BEGIN
   Zulauf_AR_Niv.Status.BA_Nrm := TRUE;
   Zulauf_AR_Niv.Status.BA_Frz := FALSE;
   Zulauf_AR_Niv.Status.BA_EW := FALSE;
   Zulauf_AR_Niv.Status.BA_Sim := FALSE;
   Zulauf_AR_Niv.Status.BA_Wart := FALSE;
   Zulauf_AR_Niv.Status.Frg_HH := FALSE;
   Zulauf_AR_Niv.Status.Frg_H := FALSE;
   Zulauf_AR_Niv.Status.Frg_L := FALSE;
   Zulauf_AR_Niv.Status.Frg_LL := FALSE;
   Zulauf_AR_Niv.Status.SB_MW_frz := FALSE;
   Zulauf_AR_Niv.Status.SB_MW_EW := FALSE;
   Zulauf_AR_Niv.Status.BM_MW_ok := TRUE;
   Zulauf_AR_Niv.Status.BM_MW_frz := FALSE;
   Zulauf_AR_Niv.Status.BM_MW_EW := FALSE;
   Zulauf_AR_Niv.Status.BM_MW_Sim := FALSE;
   Zulauf_AR_Niv.Status.BM_MW_nok := FALSE;
   Zulauf_AR_Niv.Status.BM_MW_zw := FALSE;
   Zulauf_AR_Niv.Status.GW_Sp_H := FALSE;
   Zulauf_AR_Niv.Status.GW_Sp_L := FALSE;
   Zulauf_AR_Niv.Status.Res_19 := FALSE;
   Zulauf_AR_Niv.Status.Res_26 := FALSE;
   Zulauf_AR_Niv.Status.Res_27 := FALSE;
   Zulauf_AR_Niv.Status.Res_28 := FALSE;
   Zulauf_AR_Niv.Status.Res_29 := FALSE;
   Zulauf_AR_Niv.Status.Res_30 := FALSE;
   Zulauf_AR_Niv.Status.Res_31 := FALSE;
   Zulauf_AR_Niv.Status.Res_32 := FALSE;
   Zulauf_AR_Niv.Status.Res_33 := FALSE;
   Zulauf_AR_Niv.Status.Res_34 := FALSE;
   Zulauf_AR_Niv.Status.BB_AutoOk := TRUE;
   Zulauf_AR_Niv.Status.BB_SS := FALSE;
   Zulauf_AR_Niv.Status.BB_SSnq := FALSE;
   Zulauf_AR_Niv.Stoerung.St_allg := FALSE;
   Zulauf_AR_Niv.Stoerung.St_4mA := FALSE;
   Zulauf_AR_Niv.Stoerung.St_OF := FALSE;
   Zulauf_AR_Niv.Stoerung.St_UF := FALSE;
   Zulauf_AR_Niv.Stoerung.St_Kom_DP := FALSE;
   Zulauf_AR_Niv.Stoerung.St_Kom_int := FALSE;
   Zulauf_AR_Niv.Stoerung.St_int := FALSE;
   Zulauf_AR_Niv.Stoerung.Res_7 := FALSE;
   Zulauf_AR_Niv.Stoerung.GW_HH := FALSE;
   Zulauf_AR_Niv.Stoerung.GW_H := FALSE;
   Zulauf_AR_Niv.Stoerung.GW_L := FALSE;
   Zulauf_AR_Niv.Stoerung.GW_LL := FALSE;
   Zulauf_AR_Niv.Stoerung.Res_12 := FALSE;
   Zulauf_AR_Niv.Stoerung.Res_13 := FALSE;
   Zulauf_AR_Niv.Stoerung.Res_14 := FALSE;
   Zulauf_AR_Niv.Stoerung.Res_15 := FALSE;
   Zulauf_AR_Niv.Stoerung.Res_16 := FALSE;
   Zulauf_AR_Niv.Stoerung.Res_17 := FALSE;
   Zulauf_AR_Niv.Stoerung.Res_18 := FALSE;
   Zulauf_AR_Niv.Stoerung.Res_19 := FALSE;
   Zulauf_AR_Niv.Stoerung.Res_20 := FALSE;
   Zulauf_AR_Niv.Stoerung.Res_21 := FALSE;
   Zulauf_AR_Niv.Stoerung.Res_22 := FALSE;
   Zulauf_AR_Niv.Stoerung.Res_23 := FALSE;
   Zulauf_AR_Niv.Stoerung.Res_24 := FALSE;
   Zulauf_AR_Niv.Stoerung.Res_25 := FALSE;
   Zulauf_AR_Niv.Stoerung.Res_26 := FALSE;
   Zulauf_AR_Niv.Stoerung.Res_27 := FALSE;
   Zulauf_AR_Niv.Stoerung.Res_28 := FALSE;
   Zulauf_AR_Niv.Stoerung.Res_29 := FALSE;
   Zulauf_AR_Niv.Stoerung.Res_30 := FALSE;
   Zulauf_AR_Niv.Stoerung.Res_31 := FALSE;
   Zulauf_AR_Niv.MW_akt := 21.85904;
   Zulauf_AR_Temp.Status.BA_Nrm := TRUE;
   Zulauf_AR_Temp.Status.BA_Frz := FALSE;
   Zulauf_AR_Temp.Status.BA_EW := FALSE;
   Zulauf_AR_Temp.Status.BA_Sim := FALSE;
   Zulauf_AR_Temp.Status.BA_Wart := FALSE;
   Zulauf_AR_Temp.Status.Frg_HH := FALSE;
   Zulauf_AR_Temp.Status.Frg_H := FALSE;
   Zulauf_AR_Temp.Status.Frg_L := FALSE;
   Zulauf_AR_Temp.Status.Frg_LL := FALSE;
   Zulauf_AR_Temp.Status.SB_MW_frz := FALSE;
   Zulauf_AR_Temp.Status.SB_MW_EW := FALSE;
   Zulauf_AR_Temp.Status.BM_MW_ok := TRUE;
   Zulauf_AR_Temp.Status.BM_MW_frz := FALSE;
   Zulauf_AR_Temp.Status.BM_MW_EW := FALSE;
   Zulauf_AR_Temp.Status.BM_MW_Sim := FALSE;
   Zulauf_AR_Temp.Status.BM_MW_nok := FALSE;
   Zulauf_AR_Temp.Status.BM_MW_zw := FALSE;
   Zulauf_AR_Temp.Status.GW_Sp_H := FALSE;
   Zulauf_AR_Temp.Status.GW_Sp_L := FALSE;
   Zulauf_AR_Temp.Status.Res_19 := FALSE;
   Zulauf_AR_Temp.Status.Res_26 := FALSE;
   Zulauf_AR_Temp.Status.Res_27 := FALSE;
   Zulauf_AR_Temp.Status.Res_28 := FALSE;
   Zulauf_AR_Temp.Status.Res_29 := FALSE;
   Zulauf_AR_Temp.Status.Res_30 := FALSE;
   Zulauf_AR_Temp.Status.Res_31 := FALSE;
   Zulauf_AR_Temp.Status.Res_32 := FALSE;
   Zulauf_AR_Temp.Status.Res_33 := FALSE;
   Zulauf_AR_Temp.Status.Res_34 := FALSE;
   Zulauf_AR_Temp.Status.BB_AutoOk := TRUE;
   Zulauf_AR_Temp.Status.BB_SS := FALSE;
   Zulauf_AR_Temp.Status.BB_SSnq := FALSE;
   Zulauf_AR_Temp.Stoerung.St_allg := FALSE;
   Zulauf_AR_Temp.Stoerung.St_4mA := FALSE;
   Zulauf_AR_Temp.Stoerung.St_OF := FALSE;
   Zulauf_AR_Temp.Stoerung.St_UF := FALSE;
   Zulauf_AR_Temp.Stoerung.St_Kom_DP := FALSE;
   Zulauf_AR_Temp.Stoerung.St_Kom_int := FALSE;
   Zulauf_AR_Temp.Stoerung.St_int := FALSE;
   Zulauf_AR_Temp.Stoerung.Res_7 := FALSE;
   Zulauf_AR_Temp.Stoerung.GW_HH := FALSE;
   Zulauf_AR_Temp.Stoerung.GW_H := FALSE;
   Zulauf_AR_Temp.Stoerung.GW_L := FALSE;
   Zulauf_AR_Temp.Stoerung.GW_LL := FALSE;
   Zulauf_AR_Temp.Stoerung.Res_12 := FALSE;
   Zulauf_AR_Temp.Stoerung.Res_13 := FALSE;
   Zulauf_AR_Temp.Stoerung.Res_14 := FALSE;
   Zulauf_AR_Temp.Stoerung.Res_15 := FALSE;
   Zulauf_AR_Temp.Stoerung.Res_16 := FALSE;
   Zulauf_AR_Temp.Stoerung.Res_17 := FALSE;
   Zulauf_AR_Temp.Stoerung.Res_18 := FALSE;
   Zulauf_AR_Temp.Stoerung.Res_19 := FALSE;
   Zulauf_AR_Temp.Stoerung.Res_20 := FALSE;
   Zulauf_AR_Temp.Stoerung.Res_21 := FALSE;
   Zulauf_AR_Temp.Stoerung.Res_22 := FALSE;
   Zulauf_AR_Temp.Stoerung.Res_23 := FALSE;
   Zulauf_AR_Temp.Stoerung.Res_24 := FALSE;
   Zulauf_AR_Temp.Stoerung.Res_25 := FALSE;
   Zulauf_AR_Temp.Stoerung.Res_26 := FALSE;
   Zulauf_AR_Temp.Stoerung.Res_27 := FALSE;
   Zulauf_AR_Temp.Stoerung.Res_28 := FALSE;
   Zulauf_AR_Temp.Stoerung.Res_29 := FALSE;
   Zulauf_AR_Temp.Stoerung.Res_30 := FALSE;
   Zulauf_AR_Temp.Stoerung.Res_31 := FALSE;
   Zulauf_AR_Temp.MW_akt := 0.0;
   Zulauf_AR_DF.Status.BA_Nrm := TRUE;
   Zulauf_AR_DF.Status.BA_Frz := FALSE;
   Zulauf_AR_DF.Status.BA_EW := FALSE;
   Zulauf_AR_DF.Status.BA_Sim := FALSE;
   Zulauf_AR_DF.Status.BA_Wart := FALSE;
   Zulauf_AR_DF.Status.Frg_HH := FALSE;
   Zulauf_AR_DF.Status.Frg_H := FALSE;
   Zulauf_AR_DF.Status.Frg_L := FALSE;
   Zulauf_AR_DF.Status.Frg_LL := FALSE;
   Zulauf_AR_DF.Status.SB_MW_frz := FALSE;
   Zulauf_AR_DF.Status.SB_MW_EW := FALSE;
   Zulauf_AR_DF.Status.BM_MW_ok := FALSE;
   Zulauf_AR_DF.Status.BM_MW_frz := TRUE;
   Zulauf_AR_DF.Status.BM_MW_EW := FALSE;
   Zulauf_AR_DF.Status.BM_MW_Sim := FALSE;
   Zulauf_AR_DF.Status.BM_MW_nok := TRUE;
   Zulauf_AR_DF.Status.BM_MW_zw := FALSE;
   Zulauf_AR_DF.Status.GW_Sp_H := FALSE;
   Zulauf_AR_DF.Status.GW_Sp_L := FALSE;
   Zulauf_AR_DF.Status.Res_19 := FALSE;
   Zulauf_AR_DF.Status.Res_26 := FALSE;
   Zulauf_AR_DF.Status.Res_27 := FALSE;
   Zulauf_AR_DF.Status.Res_28 := FALSE;
   Zulauf_AR_DF.Status.Res_29 := FALSE;
   Zulauf_AR_DF.Status.Res_30 := FALSE;
   Zulauf_AR_DF.Status.Res_31 := FALSE;
   Zulauf_AR_DF.Status.Res_32 := FALSE;
   Zulauf_AR_DF.Status.Res_33 := FALSE;
   Zulauf_AR_DF.Status.Res_34 := FALSE;
   Zulauf_AR_DF.Status.BB_AutoOk := FALSE;
   Zulauf_AR_DF.Status.BB_SS := TRUE;
   Zulauf_AR_DF.Status.BB_SSnq := FALSE;
   Zulauf_AR_DF.Stoerung.St_allg := FALSE;
   Zulauf_AR_DF.Stoerung.St_4mA := TRUE;
   Zulauf_AR_DF.Stoerung.St_OF := FALSE;
   Zulauf_AR_DF.Stoerung.St_UF := TRUE;
   Zulauf_AR_DF.Stoerung.St_Kom_DP := FALSE;
   Zulauf_AR_DF.Stoerung.St_Kom_int := FALSE;
   Zulauf_AR_DF.Stoerung.St_int := FALSE;
   Zulauf_AR_DF.Stoerung.Res_7 := FALSE;
   Zulauf_AR_DF.Stoerung.GW_HH := FALSE;
   Zulauf_AR_DF.Stoerung.GW_H := FALSE;
   Zulauf_AR_DF.Stoerung.GW_L := FALSE;
   Zulauf_AR_DF.Stoerung.GW_LL := FALSE;
   Zulauf_AR_DF.Stoerung.Res_12 := FALSE;
   Zulauf_AR_DF.Stoerung.Res_13 := FALSE;
   Zulauf_AR_DF.Stoerung.Res_14 := FALSE;
   Zulauf_AR_DF.Stoerung.Res_15 := FALSE;
   Zulauf_AR_DF.Stoerung.Res_16 := FALSE;
   Zulauf_AR_DF.Stoerung.Res_17 := FALSE;
   Zulauf_AR_DF.Stoerung.Res_18 := FALSE;
   Zulauf_AR_DF.Stoerung.Res_19 := FALSE;
   Zulauf_AR_DF.Stoerung.Res_20 := FALSE;
   Zulauf_AR_DF.Stoerung.Res_21 := FALSE;
   Zulauf_AR_DF.Stoerung.Res_22 := FALSE;
   Zulauf_AR_DF.Stoerung.Res_23 := FALSE;
   Zulauf_AR_DF.Stoerung.Res_24 := FALSE;
   Zulauf_AR_DF.Stoerung.Res_25 := FALSE;
   Zulauf_AR_DF.Stoerung.Res_26 := FALSE;
   Zulauf_AR_DF.Stoerung.Res_27 := FALSE;
   Zulauf_AR_DF.Stoerung.Res_28 := FALSE;
   Zulauf_AR_DF.Stoerung.Res_29 := FALSE;
   Zulauf_AR_DF.Stoerung.Res_30 := FALSE;
   Zulauf_AR_DF.Stoerung.Res_31 := FALSE;
   Zulauf_AR_DF.MW_akt := 0.0;
   BB1_AS1_SS.Status.BA_Nrm := TRUE;
   BB1_AS1_SS.Status.BA_Frz := FALSE;
   BB1_AS1_SS.Status.BA_EW := FALSE;
   BB1_AS1_SS.Status.BA_Sim := FALSE;
   BB1_AS1_SS.Status.BA_Wart := FALSE;
   BB1_AS1_SS.Status.Frg_HH := FALSE;
   BB1_AS1_SS.Status.Frg_H := FALSE;
   BB1_AS1_SS.Status.Frg_L := FALSE;
   BB1_AS1_SS.Status.Frg_LL := FALSE;
   BB1_AS1_SS.Status.SB_MW_frz := FALSE;
   BB1_AS1_SS.Status.SB_MW_EW := FALSE;
   BB1_AS1_SS.Status.BM_MW_ok := TRUE;
   BB1_AS1_SS.Status.BM_MW_frz := FALSE;
   BB1_AS1_SS.Status.BM_MW_EW := FALSE;
   BB1_AS1_SS.Status.BM_MW_Sim := FALSE;
   BB1_AS1_SS.Status.BM_MW_nok := FALSE;
   BB1_AS1_SS.Status.BM_MW_zw := FALSE;
   BB1_AS1_SS.Status.GW_Sp_H := FALSE;
   BB1_AS1_SS.Status.GW_Sp_L := FALSE;
   BB1_AS1_SS.Status.Res_19 := FALSE;
   BB1_AS1_SS.Status.Res_26 := FALSE;
   BB1_AS1_SS.Status.Res_27 := FALSE;
   BB1_AS1_SS.Status.Res_28 := FALSE;
   BB1_AS1_SS.Status.Res_29 := FALSE;
   BB1_AS1_SS.Status.Res_30 := FALSE;
   BB1_AS1_SS.Status.Res_31 := FALSE;
   BB1_AS1_SS.Status.Res_32 := FALSE;
   BB1_AS1_SS.Status.Res_33 := FALSE;
   BB1_AS1_SS.Status.Res_34 := FALSE;
   BB1_AS1_SS.Status.BB_AutoOk := TRUE;
   BB1_AS1_SS.Status.BB_SS := FALSE;
   BB1_AS1_SS.Status.BB_SSnq := FALSE;
   BB1_AS1_SS.Stoerung.St_allg := FALSE;
   BB1_AS1_SS.Stoerung.St_4mA := FALSE;
   BB1_AS1_SS.Stoerung.St_OF := FALSE;
   BB1_AS1_SS.Stoerung.St_UF := FALSE;
   BB1_AS1_SS.Stoerung.St_Kom_DP := FALSE;
   BB1_AS1_SS.Stoerung.St_Kom_int := FALSE;
   BB1_AS1_SS.Stoerung.St_int := FALSE;
   BB1_AS1_SS.Stoerung.Res_7 := FALSE;
   BB1_AS1_SS.Stoerung.GW_HH := FALSE;
   BB1_AS1_SS.Stoerung.GW_H := FALSE;
   BB1_AS1_SS.Stoerung.GW_L := FALSE;
   BB1_AS1_SS.Stoerung.GW_LL := FALSE;
   BB1_AS1_SS.Stoerung.Res_12 := FALSE;
   BB1_AS1_SS.Stoerung.Res_13 := FALSE;
   BB1_AS1_SS.Stoerung.Res_14 := FALSE;
   BB1_AS1_SS.Stoerung.Res_15 := FALSE;
   BB1_AS1_SS.Stoerung.Res_16 := FALSE;
   BB1_AS1_SS.Stoerung.Res_17 := FALSE;
   BB1_AS1_SS.Stoerung.Res_18 := FALSE;
   BB1_AS1_SS.Stoerung.Res_19 := FALSE;
   BB1_AS1_SS.Stoerung.Res_20 := FALSE;
   BB1_AS1_SS.Stoerung.Res_21 := FALSE;
   BB1_AS1_SS.Stoerung.Res_22 := FALSE;
   BB1_AS1_SS.Stoerung.Res_23 := FALSE;
   BB1_AS1_SS.Stoerung.Res_24 := FALSE;
   BB1_AS1_SS.Stoerung.Res_25 := FALSE;
   BB1_AS1_SS.Stoerung.Res_26 := FALSE;
   BB1_AS1_SS.Stoerung.Res_27 := FALSE;
   BB1_AS1_SS.Stoerung.Res_28 := FALSE;
   BB1_AS1_SS.Stoerung.Res_29 := FALSE;
   BB1_AS1_SS.Stoerung.Res_30 := FALSE;
   BB1_AS1_SS.Stoerung.Res_31 := FALSE;
   BB1_AS1_SS.MW_akt := 0.0;
   BB1_AS2_SS.Status.BA_Nrm := TRUE;
   BB1_AS2_SS.Status.BA_Frz := FALSE;
   BB1_AS2_SS.Status.BA_EW := FALSE;
   BB1_AS2_SS.Status.BA_Sim := FALSE;
   BB1_AS2_SS.Status.BA_Wart := FALSE;
   BB1_AS2_SS.Status.Frg_HH := FALSE;
   BB1_AS2_SS.Status.Frg_H := FALSE;
   BB1_AS2_SS.Status.Frg_L := FALSE;
   BB1_AS2_SS.Status.Frg_LL := FALSE;
   BB1_AS2_SS.Status.SB_MW_frz := FALSE;
   BB1_AS2_SS.Status.SB_MW_EW := FALSE;
   BB1_AS2_SS.Status.BM_MW_ok := TRUE;
   BB1_AS2_SS.Status.BM_MW_frz := FALSE;
   BB1_AS2_SS.Status.BM_MW_EW := FALSE;
   BB1_AS2_SS.Status.BM_MW_Sim := FALSE;
   BB1_AS2_SS.Status.BM_MW_nok := FALSE;
   BB1_AS2_SS.Status.BM_MW_zw := FALSE;
   BB1_AS2_SS.Status.GW_Sp_H := FALSE;
   BB1_AS2_SS.Status.GW_Sp_L := FALSE;
   BB1_AS2_SS.Status.Res_19 := FALSE;
   BB1_AS2_SS.Status.Res_26 := FALSE;
   BB1_AS2_SS.Status.Res_27 := FALSE;
   BB1_AS2_SS.Status.Res_28 := FALSE;
   BB1_AS2_SS.Status.Res_29 := FALSE;
   BB1_AS2_SS.Status.Res_30 := FALSE;
   BB1_AS2_SS.Status.Res_31 := FALSE;
   BB1_AS2_SS.Status.Res_32 := FALSE;
   BB1_AS2_SS.Status.Res_33 := FALSE;
   BB1_AS2_SS.Status.Res_34 := FALSE;
   BB1_AS2_SS.Status.BB_AutoOk := TRUE;
   BB1_AS2_SS.Status.BB_SS := FALSE;
   BB1_AS2_SS.Status.BB_SSnq := FALSE;
   BB1_AS2_SS.Stoerung.St_allg := FALSE;
   BB1_AS2_SS.Stoerung.St_4mA := FALSE;
   BB1_AS2_SS.Stoerung.St_OF := FALSE;
   BB1_AS2_SS.Stoerung.St_UF := FALSE;
   BB1_AS2_SS.Stoerung.St_Kom_DP := FALSE;
   BB1_AS2_SS.Stoerung.St_Kom_int := FALSE;
   BB1_AS2_SS.Stoerung.St_int := FALSE;
   BB1_AS2_SS.Stoerung.Res_7 := FALSE;
   BB1_AS2_SS.Stoerung.GW_HH := FALSE;
   BB1_AS2_SS.Stoerung.GW_H := FALSE;
   BB1_AS2_SS.Stoerung.GW_L := FALSE;
   BB1_AS2_SS.Stoerung.GW_LL := FALSE;
   BB1_AS2_SS.Stoerung.Res_12 := FALSE;
   BB1_AS2_SS.Stoerung.Res_13 := FALSE;
   BB1_AS2_SS.Stoerung.Res_14 := FALSE;
   BB1_AS2_SS.Stoerung.Res_15 := FALSE;
   BB1_AS2_SS.Stoerung.Res_16 := FALSE;
   BB1_AS2_SS.Stoerung.Res_17 := FALSE;
   BB1_AS2_SS.Stoerung.Res_18 := FALSE;
   BB1_AS2_SS.Stoerung.Res_19 := FALSE;
   BB1_AS2_SS.Stoerung.Res_20 := FALSE;
   BB1_AS2_SS.Stoerung.Res_21 := FALSE;
   BB1_AS2_SS.Stoerung.Res_22 := FALSE;
   BB1_AS2_SS.Stoerung.Res_23 := FALSE;
   BB1_AS2_SS.Stoerung.Res_24 := FALSE;
   BB1_AS2_SS.Stoerung.Res_25 := FALSE;
   BB1_AS2_SS.Stoerung.Res_26 := FALSE;
   BB1_AS2_SS.Stoerung.Res_27 := FALSE;
   BB1_AS2_SS.Stoerung.Res_28 := FALSE;
   BB1_AS2_SS.Stoerung.Res_29 := FALSE;
   BB1_AS2_SS.Stoerung.Res_30 := FALSE;
   BB1_AS2_SS.Stoerung.Res_31 := FALSE;
   BB1_AS2_SS.MW_akt := 76.62236;
   BB2_AS1_SS.Status.BA_Nrm := TRUE;
   BB2_AS1_SS.Status.BA_Frz := FALSE;
   BB2_AS1_SS.Status.BA_EW := FALSE;
   BB2_AS1_SS.Status.BA_Sim := FALSE;
   BB2_AS1_SS.Status.BA_Wart := FALSE;
   BB2_AS1_SS.Status.Frg_HH := FALSE;
   BB2_AS1_SS.Status.Frg_H := FALSE;
   BB2_AS1_SS.Status.Frg_L := FALSE;
   BB2_AS1_SS.Status.Frg_LL := FALSE;
   BB2_AS1_SS.Status.SB_MW_frz := FALSE;
   BB2_AS1_SS.Status.SB_MW_EW := FALSE;
   BB2_AS1_SS.Status.BM_MW_ok := TRUE;
   BB2_AS1_SS.Status.BM_MW_frz := FALSE;
   BB2_AS1_SS.Status.BM_MW_EW := FALSE;
   BB2_AS1_SS.Status.BM_MW_Sim := FALSE;
   BB2_AS1_SS.Status.BM_MW_nok := FALSE;
   BB2_AS1_SS.Status.BM_MW_zw := FALSE;
   BB2_AS1_SS.Status.GW_Sp_H := FALSE;
   BB2_AS1_SS.Status.GW_Sp_L := FALSE;
   BB2_AS1_SS.Status.Res_19 := FALSE;
   BB2_AS1_SS.Status.Res_26 := FALSE;
   BB2_AS1_SS.Status.Res_27 := FALSE;
   BB2_AS1_SS.Status.Res_28 := FALSE;
   BB2_AS1_SS.Status.Res_29 := FALSE;
   BB2_AS1_SS.Status.Res_30 := FALSE;
   BB2_AS1_SS.Status.Res_31 := FALSE;
   BB2_AS1_SS.Status.Res_32 := FALSE;
   BB2_AS1_SS.Status.Res_33 := FALSE;
   BB2_AS1_SS.Status.Res_34 := FALSE;
   BB2_AS1_SS.Status.BB_AutoOk := TRUE;
   BB2_AS1_SS.Status.BB_SS := FALSE;
   BB2_AS1_SS.Status.BB_SSnq := FALSE;
   BB2_AS1_SS.Stoerung.St_allg := FALSE;
   BB2_AS1_SS.Stoerung.St_4mA := FALSE;
   BB2_AS1_SS.Stoerung.St_OF := FALSE;
   BB2_AS1_SS.Stoerung.St_UF := FALSE;
   BB2_AS1_SS.Stoerung.St_Kom_DP := FALSE;
   BB2_AS1_SS.Stoerung.St_Kom_int := FALSE;
   BB2_AS1_SS.Stoerung.St_int := FALSE;
   BB2_AS1_SS.Stoerung.Res_7 := FALSE;
   BB2_AS1_SS.Stoerung.GW_HH := FALSE;
   BB2_AS1_SS.Stoerung.GW_H := FALSE;
   BB2_AS1_SS.Stoerung.GW_L := FALSE;
   BB2_AS1_SS.Stoerung.GW_LL := FALSE;
   BB2_AS1_SS.Stoerung.Res_12 := FALSE;
   BB2_AS1_SS.Stoerung.Res_13 := FALSE;
   BB2_AS1_SS.Stoerung.Res_14 := FALSE;
   BB2_AS1_SS.Stoerung.Res_15 := FALSE;
   BB2_AS1_SS.Stoerung.Res_16 := FALSE;
   BB2_AS1_SS.Stoerung.Res_17 := FALSE;
   BB2_AS1_SS.Stoerung.Res_18 := FALSE;
   BB2_AS1_SS.Stoerung.Res_19 := FALSE;
   BB2_AS1_SS.Stoerung.Res_20 := FALSE;
   BB2_AS1_SS.Stoerung.Res_21 := FALSE;
   BB2_AS1_SS.Stoerung.Res_22 := FALSE;
   BB2_AS1_SS.Stoerung.Res_23 := FALSE;
   BB2_AS1_SS.Stoerung.Res_24 := FALSE;
   BB2_AS1_SS.Stoerung.Res_25 := FALSE;
   BB2_AS1_SS.Stoerung.Res_26 := FALSE;
   BB2_AS1_SS.Stoerung.Res_27 := FALSE;
   BB2_AS1_SS.Stoerung.Res_28 := FALSE;
   BB2_AS1_SS.Stoerung.Res_29 := FALSE;
   BB2_AS1_SS.Stoerung.Res_30 := FALSE;
   BB2_AS1_SS.Stoerung.Res_31 := FALSE;
   BB2_AS1_SS.MW_akt := 0.05018311;
   BB2_AS2_SS.Status.BA_Nrm := TRUE;
   BB2_AS2_SS.Status.BA_Frz := FALSE;
   BB2_AS2_SS.Status.BA_EW := FALSE;
   BB2_AS2_SS.Status.BA_Sim := FALSE;
   BB2_AS2_SS.Status.BA_Wart := FALSE;
   BB2_AS2_SS.Status.Frg_HH := FALSE;
   BB2_AS2_SS.Status.Frg_H := FALSE;
   BB2_AS2_SS.Status.Frg_L := FALSE;
   BB2_AS2_SS.Status.Frg_LL := FALSE;
   BB2_AS2_SS.Status.SB_MW_frz := FALSE;
   BB2_AS2_SS.Status.SB_MW_EW := FALSE;
   BB2_AS2_SS.Status.BM_MW_ok := TRUE;
   BB2_AS2_SS.Status.BM_MW_frz := FALSE;
   BB2_AS2_SS.Status.BM_MW_EW := FALSE;
   BB2_AS2_SS.Status.BM_MW_Sim := FALSE;
   BB2_AS2_SS.Status.BM_MW_nok := FALSE;
   BB2_AS2_SS.Status.BM_MW_zw := FALSE;
   BB2_AS2_SS.Status.GW_Sp_H := FALSE;
   BB2_AS2_SS.Status.GW_Sp_L := FALSE;
   BB2_AS2_SS.Status.Res_19 := FALSE;
   BB2_AS2_SS.Status.Res_26 := FALSE;
   BB2_AS2_SS.Status.Res_27 := FALSE;
   BB2_AS2_SS.Status.Res_28 := FALSE;
   BB2_AS2_SS.Status.Res_29 := FALSE;
   BB2_AS2_SS.Status.Res_30 := FALSE;
   BB2_AS2_SS.Status.Res_31 := FALSE;
   BB2_AS2_SS.Status.Res_32 := FALSE;
   BB2_AS2_SS.Status.Res_33 := FALSE;
   BB2_AS2_SS.Status.Res_34 := FALSE;
   BB2_AS2_SS.Status.BB_AutoOk := TRUE;
   BB2_AS2_SS.Status.BB_SS := FALSE;
   BB2_AS2_SS.Status.BB_SSnq := FALSE;
   BB2_AS2_SS.Stoerung.St_allg := FALSE;
   BB2_AS2_SS.Stoerung.St_4mA := FALSE;
   BB2_AS2_SS.Stoerung.St_OF := FALSE;
   BB2_AS2_SS.Stoerung.St_UF := FALSE;
   BB2_AS2_SS.Stoerung.St_Kom_DP := FALSE;
   BB2_AS2_SS.Stoerung.St_Kom_int := FALSE;
   BB2_AS2_SS.Stoerung.St_int := FALSE;
   BB2_AS2_SS.Stoerung.Res_7 := FALSE;
   BB2_AS2_SS.Stoerung.GW_HH := FALSE;
   BB2_AS2_SS.Stoerung.GW_H := FALSE;
   BB2_AS2_SS.Stoerung.GW_L := FALSE;
   BB2_AS2_SS.Stoerung.GW_LL := FALSE;
   BB2_AS2_SS.Stoerung.Res_12 := FALSE;
   BB2_AS2_SS.Stoerung.Res_13 := FALSE;
   BB2_AS2_SS.Stoerung.Res_14 := FALSE;
   BB2_AS2_SS.Stoerung.Res_15 := FALSE;
   BB2_AS2_SS.Stoerung.Res_16 := FALSE;
   BB2_AS2_SS.Stoerung.Res_17 := FALSE;
   BB2_AS2_SS.Stoerung.Res_18 := FALSE;
   BB2_AS2_SS.Stoerung.Res_19 := FALSE;
   BB2_AS2_SS.Stoerung.Res_20 := FALSE;
   BB2_AS2_SS.Stoerung.Res_21 := FALSE;
   BB2_AS2_SS.Stoerung.Res_22 := FALSE;
   BB2_AS2_SS.Stoerung.Res_23 := FALSE;
   BB2_AS2_SS.Stoerung.Res_24 := FALSE;
   BB2_AS2_SS.Stoerung.Res_25 := FALSE;
   BB2_AS2_SS.Stoerung.Res_26 := FALSE;
   BB2_AS2_SS.Stoerung.Res_27 := FALSE;
   BB2_AS2_SS.Stoerung.Res_28 := FALSE;
   BB2_AS2_SS.Stoerung.Res_29 := FALSE;
   BB2_AS2_SS.Stoerung.Res_30 := FALSE;
   BB2_AS2_SS.Stoerung.Res_31 := FALSE;
   BB2_AS2_SS.MW_akt := 0.140151;
   BB1_O2.Status.BA_Nrm := TRUE;
   BB1_O2.Status.BA_Frz := FALSE;
   BB1_O2.Status.BA_EW := FALSE;
   BB1_O2.Status.BA_Sim := FALSE;
   BB1_O2.Status.BA_Wart := FALSE;
   BB1_O2.Status.Frg_HH := FALSE;
   BB1_O2.Status.Frg_H := FALSE;
   BB1_O2.Status.Frg_L := FALSE;
   BB1_O2.Status.Frg_LL := TRUE;
   BB1_O2.Status.SB_MW_frz := FALSE;
   BB1_O2.Status.SB_MW_EW := FALSE;
   BB1_O2.Status.BM_MW_ok := TRUE;
   BB1_O2.Status.BM_MW_frz := FALSE;
   BB1_O2.Status.BM_MW_EW := FALSE;
   BB1_O2.Status.BM_MW_Sim := FALSE;
   BB1_O2.Status.BM_MW_nok := FALSE;
   BB1_O2.Status.BM_MW_zw := FALSE;
   BB1_O2.Status.GW_Sp_H := FALSE;
   BB1_O2.Status.GW_Sp_L := FALSE;
   BB1_O2.Status.Res_19 := FALSE;
   BB1_O2.Status.Res_26 := FALSE;
   BB1_O2.Status.Res_27 := FALSE;
   BB1_O2.Status.Res_28 := FALSE;
   BB1_O2.Status.Res_29 := FALSE;
   BB1_O2.Status.Res_30 := FALSE;
   BB1_O2.Status.Res_31 := FALSE;
   BB1_O2.Status.Res_32 := FALSE;
   BB1_O2.Status.Res_33 := FALSE;
   BB1_O2.Status.Res_34 := FALSE;
   BB1_O2.Status.BB_AutoOk := TRUE;
   BB1_O2.Status.BB_SS := FALSE;
   BB1_O2.Status.BB_SSnq := FALSE;
   BB1_O2.Stoerung.St_allg := FALSE;
   BB1_O2.Stoerung.St_4mA := FALSE;
   BB1_O2.Stoerung.St_OF := FALSE;
   BB1_O2.Stoerung.St_UF := FALSE;
   BB1_O2.Stoerung.St_Kom_DP := FALSE;
   BB1_O2.Stoerung.St_Kom_int := FALSE;
   BB1_O2.Stoerung.St_int := FALSE;
   BB1_O2.Stoerung.Res_7 := FALSE;
   BB1_O2.Stoerung.GW_HH := FALSE;
   BB1_O2.Stoerung.GW_H := FALSE;
   BB1_O2.Stoerung.GW_L := FALSE;
   BB1_O2.Stoerung.GW_LL := FALSE;
   BB1_O2.Stoerung.Res_12 := FALSE;
   BB1_O2.Stoerung.Res_13 := FALSE;
   BB1_O2.Stoerung.Res_14 := FALSE;
   BB1_O2.Stoerung.Res_15 := FALSE;
   BB1_O2.Stoerung.Res_16 := FALSE;
   BB1_O2.Stoerung.Res_17 := FALSE;
   BB1_O2.Stoerung.Res_18 := FALSE;
   BB1_O2.Stoerung.Res_19 := FALSE;
   BB1_O2.Stoerung.Res_20 := FALSE;
   BB1_O2.Stoerung.Res_21 := FALSE;
   BB1_O2.Stoerung.Res_22 := FALSE;
   BB1_O2.Stoerung.Res_23 := FALSE;
   BB1_O2.Stoerung.Res_24 := FALSE;
   BB1_O2.Stoerung.Res_25 := FALSE;
   BB1_O2.Stoerung.Res_26 := FALSE;
   BB1_O2.Stoerung.Res_27 := FALSE;
   BB1_O2.Stoerung.Res_28 := FALSE;
   BB1_O2.Stoerung.Res_29 := FALSE;
   BB1_O2.Stoerung.Res_30 := FALSE;
   BB1_O2.Stoerung.Res_31 := FALSE;
   BB1_O2.MW_akt := 1.563633;
   BB1_Temp.Status.BA_Nrm := TRUE;
   BB1_Temp.Status.BA_Frz := FALSE;
   BB1_Temp.Status.BA_EW := FALSE;
   BB1_Temp.Status.BA_Sim := FALSE;
   BB1_Temp.Status.BA_Wart := FALSE;
   BB1_Temp.Status.Frg_HH := FALSE;
   BB1_Temp.Status.Frg_H := FALSE;
   BB1_Temp.Status.Frg_L := FALSE;
   BB1_Temp.Status.Frg_LL := FALSE;
   BB1_Temp.Status.SB_MW_frz := FALSE;
   BB1_Temp.Status.SB_MW_EW := FALSE;
   BB1_Temp.Status.BM_MW_ok := TRUE;
   BB1_Temp.Status.BM_MW_frz := FALSE;
   BB1_Temp.Status.BM_MW_EW := FALSE;
   BB1_Temp.Status.BM_MW_Sim := FALSE;
   BB1_Temp.Status.BM_MW_nok := FALSE;
   BB1_Temp.Status.BM_MW_zw := FALSE;
   BB1_Temp.Status.GW_Sp_H := FALSE;
   BB1_Temp.Status.GW_Sp_L := FALSE;
   BB1_Temp.Status.Res_19 := FALSE;
   BB1_Temp.Status.Res_26 := FALSE;
   BB1_Temp.Status.Res_27 := FALSE;
   BB1_Temp.Status.Res_28 := FALSE;
   BB1_Temp.Status.Res_29 := FALSE;
   BB1_Temp.Status.Res_30 := FALSE;
   BB1_Temp.Status.Res_31 := FALSE;
   BB1_Temp.Status.Res_32 := FALSE;
   BB1_Temp.Status.Res_33 := FALSE;
   BB1_Temp.Status.Res_34 := FALSE;
   BB1_Temp.Status.BB_AutoOk := TRUE;
   BB1_Temp.Status.BB_SS := FALSE;
   BB1_Temp.Status.BB_SSnq := FALSE;
   BB1_Temp.Stoerung.St_allg := FALSE;
   BB1_Temp.Stoerung.St_4mA := FALSE;
   BB1_Temp.Stoerung.St_OF := FALSE;
   BB1_Temp.Stoerung.St_UF := FALSE;
   BB1_Temp.Stoerung.St_Kom_DP := FALSE;
   BB1_Temp.Stoerung.St_Kom_int := FALSE;
   BB1_Temp.Stoerung.St_int := FALSE;
   BB1_Temp.Stoerung.Res_7 := FALSE;
   BB1_Temp.Stoerung.GW_HH := FALSE;
   BB1_Temp.Stoerung.GW_H := FALSE;
   BB1_Temp.Stoerung.GW_L := FALSE;
   BB1_Temp.Stoerung.GW_LL := FALSE;
   BB1_Temp.Stoerung.Res_12 := FALSE;
   BB1_Temp.Stoerung.Res_13 := FALSE;
   BB1_Temp.Stoerung.Res_14 := FALSE;
   BB1_Temp.Stoerung.Res_15 := FALSE;
   BB1_Temp.Stoerung.Res_16 := FALSE;
   BB1_Temp.Stoerung.Res_17 := FALSE;
   BB1_Temp.Stoerung.Res_18 := FALSE;
   BB1_Temp.Stoerung.Res_19 := FALSE;
   BB1_Temp.Stoerung.Res_20 := FALSE;
   BB1_Temp.Stoerung.Res_21 := FALSE;
   BB1_Temp.Stoerung.Res_22 := FALSE;
   BB1_Temp.Stoerung.Res_23 := FALSE;
   BB1_Temp.Stoerung.Res_24 := FALSE;
   BB1_Temp.Stoerung.Res_25 := FALSE;
   BB1_Temp.Stoerung.Res_26 := FALSE;
   BB1_Temp.Stoerung.Res_27 := FALSE;
   BB1_Temp.Stoerung.Res_28 := FALSE;
   BB1_Temp.Stoerung.Res_29 := FALSE;
   BB1_Temp.Stoerung.Res_30 := FALSE;
   BB1_Temp.Stoerung.Res_31 := FALSE;
   BB1_Temp.MW_akt := 14.53094;
   BB2_O2.Status.BA_Nrm := TRUE;
   BB2_O2.Status.BA_Frz := FALSE;
   BB2_O2.Status.BA_EW := FALSE;
   BB2_O2.Status.BA_Sim := FALSE;
   BB2_O2.Status.BA_Wart := FALSE;
   BB2_O2.Status.Frg_HH := FALSE;
   BB2_O2.Status.Frg_H := FALSE;
   BB2_O2.Status.Frg_L := FALSE;
   BB2_O2.Status.Frg_LL := TRUE;
   BB2_O2.Status.SB_MW_frz := FALSE;
   BB2_O2.Status.SB_MW_EW := FALSE;
   BB2_O2.Status.BM_MW_ok := TRUE;
   BB2_O2.Status.BM_MW_frz := FALSE;
   BB2_O2.Status.BM_MW_EW := FALSE;
   BB2_O2.Status.BM_MW_Sim := FALSE;
   BB2_O2.Status.BM_MW_nok := FALSE;
   BB2_O2.Status.BM_MW_zw := FALSE;
   BB2_O2.Status.GW_Sp_H := FALSE;
   BB2_O2.Status.GW_Sp_L := FALSE;
   BB2_O2.Status.Res_19 := FALSE;
   BB2_O2.Status.Res_26 := FALSE;
   BB2_O2.Status.Res_27 := FALSE;
   BB2_O2.Status.Res_28 := FALSE;
   BB2_O2.Status.Res_29 := FALSE;
   BB2_O2.Status.Res_30 := FALSE;
   BB2_O2.Status.Res_31 := FALSE;
   BB2_O2.Status.Res_32 := FALSE;
   BB2_O2.Status.Res_33 := FALSE;
   BB2_O2.Status.Res_34 := FALSE;
   BB2_O2.Status.BB_AutoOk := TRUE;
   BB2_O2.Status.BB_SS := FALSE;
   BB2_O2.Status.BB_SSnq := FALSE;
   BB2_O2.Stoerung.St_allg := FALSE;
   BB2_O2.Stoerung.St_4mA := FALSE;
   BB2_O2.Stoerung.St_OF := FALSE;
   BB2_O2.Stoerung.St_UF := FALSE;
   BB2_O2.Stoerung.St_Kom_DP := FALSE;
   BB2_O2.Stoerung.St_Kom_int := FALSE;
   BB2_O2.Stoerung.St_int := FALSE;
   BB2_O2.Stoerung.Res_7 := FALSE;
   BB2_O2.Stoerung.GW_HH := FALSE;
   BB2_O2.Stoerung.GW_H := FALSE;
   BB2_O2.Stoerung.GW_L := FALSE;
   BB2_O2.Stoerung.GW_LL := FALSE;
   BB2_O2.Stoerung.Res_12 := FALSE;
   BB2_O2.Stoerung.Res_13 := FALSE;
   BB2_O2.Stoerung.Res_14 := FALSE;
   BB2_O2.Stoerung.Res_15 := FALSE;
   BB2_O2.Stoerung.Res_16 := FALSE;
   BB2_O2.Stoerung.Res_17 := FALSE;
   BB2_O2.Stoerung.Res_18 := FALSE;
   BB2_O2.Stoerung.Res_19 := FALSE;
   BB2_O2.Stoerung.Res_20 := FALSE;
   BB2_O2.Stoerung.Res_21 := FALSE;
   BB2_O2.Stoerung.Res_22 := FALSE;
   BB2_O2.Stoerung.Res_23 := FALSE;
   BB2_O2.Stoerung.Res_24 := FALSE;
   BB2_O2.Stoerung.Res_25 := FALSE;
   BB2_O2.Stoerung.Res_26 := FALSE;
   BB2_O2.Stoerung.Res_27 := FALSE;
   BB2_O2.Stoerung.Res_28 := FALSE;
   BB2_O2.Stoerung.Res_29 := FALSE;
   BB2_O2.Stoerung.Res_30 := FALSE;
   BB2_O2.Stoerung.Res_31 := FALSE;
   BB2_O2.MW_akt := 1.491101;
   BB2_Temp.Status.BA_Nrm := TRUE;
   BB2_Temp.Status.BA_Frz := FALSE;
   BB2_Temp.Status.BA_EW := FALSE;
   BB2_Temp.Status.BA_Sim := FALSE;
   BB2_Temp.Status.BA_Wart := FALSE;
   BB2_Temp.Status.Frg_HH := FALSE;
   BB2_Temp.Status.Frg_H := FALSE;
   BB2_Temp.Status.Frg_L := FALSE;
   BB2_Temp.Status.Frg_LL := FALSE;
   BB2_Temp.Status.SB_MW_frz := FALSE;
   BB2_Temp.Status.SB_MW_EW := FALSE;
   BB2_Temp.Status.BM_MW_ok := TRUE;
   BB2_Temp.Status.BM_MW_frz := FALSE;
   BB2_Temp.Status.BM_MW_EW := FALSE;
   BB2_Temp.Status.BM_MW_Sim := FALSE;
   BB2_Temp.Status.BM_MW_nok := FALSE;
   BB2_Temp.Status.BM_MW_zw := FALSE;
   BB2_Temp.Status.GW_Sp_H := FALSE;
   BB2_Temp.Status.GW_Sp_L := FALSE;
   BB2_Temp.Status.Res_19 := FALSE;
   BB2_Temp.Status.Res_26 := FALSE;
   BB2_Temp.Status.Res_27 := FALSE;
   BB2_Temp.Status.Res_28 := FALSE;
   BB2_Temp.Status.Res_29 := FALSE;
   BB2_Temp.Status.Res_30 := FALSE;
   BB2_Temp.Status.Res_31 := FALSE;
   BB2_Temp.Status.Res_32 := FALSE;
   BB2_Temp.Status.Res_33 := FALSE;
   BB2_Temp.Status.Res_34 := FALSE;
   BB2_Temp.Status.BB_AutoOk := TRUE;
   BB2_Temp.Status.BB_SS := FALSE;
   BB2_Temp.Status.BB_SSnq := FALSE;
   BB2_Temp.Stoerung.St_allg := FALSE;
   BB2_Temp.Stoerung.St_4mA := FALSE;
   BB2_Temp.Stoerung.St_OF := FALSE;
   BB2_Temp.Stoerung.St_UF := FALSE;
   BB2_Temp.Stoerung.St_Kom_DP := FALSE;
   BB2_Temp.Stoerung.St_Kom_int := FALSE;
   BB2_Temp.Stoerung.St_int := FALSE;
   BB2_Temp.Stoerung.Res_7 := FALSE;
   BB2_Temp.Stoerung.GW_HH := FALSE;
   BB2_Temp.Stoerung.GW_H := FALSE;
   BB2_Temp.Stoerung.GW_L := FALSE;
   BB2_Temp.Stoerung.GW_LL := FALSE;
   BB2_Temp.Stoerung.Res_12 := FALSE;
   BB2_Temp.Stoerung.Res_13 := FALSE;
   BB2_Temp.Stoerung.Res_14 := FALSE;
   BB2_Temp.Stoerung.Res_15 := FALSE;
   BB2_Temp.Stoerung.Res_16 := FALSE;
   BB2_Temp.Stoerung.Res_17 := FALSE;
   BB2_Temp.Stoerung.Res_18 := FALSE;
   BB2_Temp.Stoerung.Res_19 := FALSE;
   BB2_Temp.Stoerung.Res_20 := FALSE;
   BB2_Temp.Stoerung.Res_21 := FALSE;
   BB2_Temp.Stoerung.Res_22 := FALSE;
   BB2_Temp.Stoerung.Res_23 := FALSE;
   BB2_Temp.Stoerung.Res_24 := FALSE;
   BB2_Temp.Stoerung.Res_25 := FALSE;
   BB2_Temp.Stoerung.Res_26 := FALSE;
   BB2_Temp.Stoerung.Res_27 := FALSE;
   BB2_Temp.Stoerung.Res_28 := FALSE;
   BB2_Temp.Stoerung.Res_29 := FALSE;
   BB2_Temp.Stoerung.Res_30 := FALSE;
   BB2_Temp.Stoerung.Res_31 := FALSE;
   BB2_Temp.MW_akt := 14.3844;
   BB1_DF.Status.BA_Nrm := TRUE;
   BB1_DF.Status.BA_Frz := FALSE;
   BB1_DF.Status.BA_EW := FALSE;
   BB1_DF.Status.BA_Sim := FALSE;
   BB1_DF.Status.BA_Wart := FALSE;
   BB1_DF.Status.Frg_HH := FALSE;
   BB1_DF.Status.Frg_H := FALSE;
   BB1_DF.Status.Frg_L := FALSE;
   BB1_DF.Status.Frg_LL := FALSE;
   BB1_DF.Status.SB_MW_frz := FALSE;
   BB1_DF.Status.SB_MW_EW := FALSE;
   BB1_DF.Status.BM_MW_ok := TRUE;
   BB1_DF.Status.BM_MW_frz := FALSE;
   BB1_DF.Status.BM_MW_EW := FALSE;
   BB1_DF.Status.BM_MW_Sim := FALSE;
   BB1_DF.Status.BM_MW_nok := FALSE;
   BB1_DF.Status.BM_MW_zw := FALSE;
   BB1_DF.Status.GW_Sp_H := FALSE;
   BB1_DF.Status.GW_Sp_L := FALSE;
   BB1_DF.Status.Res_19 := FALSE;
   BB1_DF.Status.Res_26 := FALSE;
   BB1_DF.Status.Res_27 := FALSE;
   BB1_DF.Status.Res_28 := FALSE;
   BB1_DF.Status.Res_29 := FALSE;
   BB1_DF.Status.Res_30 := FALSE;
   BB1_DF.Status.Res_31 := FALSE;
   BB1_DF.Status.Res_32 := FALSE;
   BB1_DF.Status.Res_33 := FALSE;
   BB1_DF.Status.Res_34 := FALSE;
   BB1_DF.Status.BB_AutoOk := TRUE;
   BB1_DF.Status.BB_SS := FALSE;
   BB1_DF.Status.BB_SSnq := FALSE;
   BB1_DF.Stoerung.St_allg := FALSE;
   BB1_DF.Stoerung.St_4mA := FALSE;
   BB1_DF.Stoerung.St_OF := FALSE;
   BB1_DF.Stoerung.St_UF := FALSE;
   BB1_DF.Stoerung.St_Kom_DP := FALSE;
   BB1_DF.Stoerung.St_Kom_int := FALSE;
   BB1_DF.Stoerung.St_int := FALSE;
   BB1_DF.Stoerung.Res_7 := FALSE;
   BB1_DF.Stoerung.GW_HH := FALSE;
   BB1_DF.Stoerung.GW_H := FALSE;
   BB1_DF.Stoerung.GW_L := FALSE;
   BB1_DF.Stoerung.GW_LL := FALSE;
   BB1_DF.Stoerung.Res_12 := FALSE;
   BB1_DF.Stoerung.Res_13 := FALSE;
   BB1_DF.Stoerung.Res_14 := FALSE;
   BB1_DF.Stoerung.Res_15 := FALSE;
   BB1_DF.Stoerung.Res_16 := FALSE;
   BB1_DF.Stoerung.Res_17 := FALSE;
   BB1_DF.Stoerung.Res_18 := FALSE;
   BB1_DF.Stoerung.Res_19 := FALSE;
   BB1_DF.Stoerung.Res_20 := FALSE;
   BB1_DF.Stoerung.Res_21 := FALSE;
   BB1_DF.Stoerung.Res_22 := FALSE;
   BB1_DF.Stoerung.Res_23 := FALSE;
   BB1_DF.Stoerung.Res_24 := FALSE;
   BB1_DF.Stoerung.Res_25 := FALSE;
   BB1_DF.Stoerung.Res_26 := FALSE;
   BB1_DF.Stoerung.Res_27 := FALSE;
   BB1_DF.Stoerung.Res_28 := FALSE;
   BB1_DF.Stoerung.Res_29 := FALSE;
   BB1_DF.Stoerung.Res_30 := FALSE;
   BB1_DF.Stoerung.Res_31 := FALSE;
   BB1_DF.MW_akt := 0.0;
   BB2_DF.Status.BA_Nrm := TRUE;
   BB2_DF.Status.BA_Frz := FALSE;
   BB2_DF.Status.BA_EW := FALSE;
   BB2_DF.Status.BA_Sim := FALSE;
   BB2_DF.Status.BA_Wart := FALSE;
   BB2_DF.Status.Frg_HH := FALSE;
   BB2_DF.Status.Frg_H := FALSE;
   BB2_DF.Status.Frg_L := FALSE;
   BB2_DF.Status.Frg_LL := FALSE;
   BB2_DF.Status.SB_MW_frz := FALSE;
   BB2_DF.Status.SB_MW_EW := FALSE;
   BB2_DF.Status.BM_MW_ok := TRUE;
   BB2_DF.Status.BM_MW_frz := FALSE;
   BB2_DF.Status.BM_MW_EW := FALSE;
   BB2_DF.Status.BM_MW_Sim := FALSE;
   BB2_DF.Status.BM_MW_nok := FALSE;
   BB2_DF.Status.BM_MW_zw := FALSE;
   BB2_DF.Status.GW_Sp_H := FALSE;
   BB2_DF.Status.GW_Sp_L := FALSE;
   BB2_DF.Status.Res_19 := FALSE;
   BB2_DF.Status.Res_26 := FALSE;
   BB2_DF.Status.Res_27 := FALSE;
   BB2_DF.Status.Res_28 := FALSE;
   BB2_DF.Status.Res_29 := FALSE;
   BB2_DF.Status.Res_30 := FALSE;
   BB2_DF.Status.Res_31 := FALSE;
   BB2_DF.Status.Res_32 := FALSE;
   BB2_DF.Status.Res_33 := FALSE;
   BB2_DF.Status.Res_34 := FALSE;
   BB2_DF.Status.BB_AutoOk := TRUE;
   BB2_DF.Status.BB_SS := FALSE;
   BB2_DF.Status.BB_SSnq := FALSE;
   BB2_DF.Stoerung.St_allg := FALSE;
   BB2_DF.Stoerung.St_4mA := FALSE;
   BB2_DF.Stoerung.St_OF := FALSE;
   BB2_DF.Stoerung.St_UF := FALSE;
   BB2_DF.Stoerung.St_Kom_DP := FALSE;
   BB2_DF.Stoerung.St_Kom_int := FALSE;
   BB2_DF.Stoerung.St_int := FALSE;
   BB2_DF.Stoerung.Res_7 := FALSE;
   BB2_DF.Stoerung.GW_HH := FALSE;
   BB2_DF.Stoerung.GW_H := FALSE;
   BB2_DF.Stoerung.GW_L := FALSE;
   BB2_DF.Stoerung.GW_LL := FALSE;
   BB2_DF.Stoerung.Res_12 := FALSE;
   BB2_DF.Stoerung.Res_13 := FALSE;
   BB2_DF.Stoerung.Res_14 := FALSE;
   BB2_DF.Stoerung.Res_15 := FALSE;
   BB2_DF.Stoerung.Res_16 := FALSE;
   BB2_DF.Stoerung.Res_17 := FALSE;
   BB2_DF.Stoerung.Res_18 := FALSE;
   BB2_DF.Stoerung.Res_19 := FALSE;
   BB2_DF.Stoerung.Res_20 := FALSE;
   BB2_DF.Stoerung.Res_21 := FALSE;
   BB2_DF.Stoerung.Res_22 := FALSE;
   BB2_DF.Stoerung.Res_23 := FALSE;
   BB2_DF.Stoerung.Res_24 := FALSE;
   BB2_DF.Stoerung.Res_25 := FALSE;
   BB2_DF.Stoerung.Res_26 := FALSE;
   BB2_DF.Stoerung.Res_27 := FALSE;
   BB2_DF.Stoerung.Res_28 := FALSE;
   BB2_DF.Stoerung.Res_29 := FALSE;
   BB2_DF.Stoerung.Res_30 := FALSE;
   BB2_DF.Stoerung.Res_31 := FALSE;
   BB2_DF.MW_akt := 0.0;
   Zulauf_Niv.Status.BA_Nrm := TRUE;
   Zulauf_Niv.Status.BA_Frz := FALSE;
   Zulauf_Niv.Status.BA_EW := FALSE;
   Zulauf_Niv.Status.BA_Sim := FALSE;
   Zulauf_Niv.Status.BA_Wart := FALSE;
   Zulauf_Niv.Status.Frg_HH := FALSE;
   Zulauf_Niv.Status.Frg_H := FALSE;
   Zulauf_Niv.Status.Frg_L := FALSE;
   Zulauf_Niv.Status.Frg_LL := FALSE;
   Zulauf_Niv.Status.SB_MW_frz := FALSE;
   Zulauf_Niv.Status.SB_MW_EW := FALSE;
   Zulauf_Niv.Status.BM_MW_ok := TRUE;
   Zulauf_Niv.Status.BM_MW_frz := FALSE;
   Zulauf_Niv.Status.BM_MW_EW := FALSE;
   Zulauf_Niv.Status.BM_MW_Sim := FALSE;
   Zulauf_Niv.Status.BM_MW_nok := FALSE;
   Zulauf_Niv.Status.BM_MW_zw := FALSE;
   Zulauf_Niv.Status.GW_Sp_H := FALSE;
   Zulauf_Niv.Status.GW_Sp_L := FALSE;
   Zulauf_Niv.Status.Res_19 := FALSE;
   Zulauf_Niv.Status.Res_26 := FALSE;
   Zulauf_Niv.Status.Res_27 := FALSE;
   Zulauf_Niv.Status.Res_28 := FALSE;
   Zulauf_Niv.Status.Res_29 := FALSE;
   Zulauf_Niv.Status.Res_30 := FALSE;
   Zulauf_Niv.Status.Res_31 := FALSE;
   Zulauf_Niv.Status.Res_32 := FALSE;
   Zulauf_Niv.Status.Res_33 := FALSE;
   Zulauf_Niv.Status.Res_34 := FALSE;
   Zulauf_Niv.Status.BB_AutoOk := TRUE;
   Zulauf_Niv.Status.BB_SS := FALSE;
   Zulauf_Niv.Status.BB_SSnq := FALSE;
   Zulauf_Niv.Stoerung.St_allg := FALSE;
   Zulauf_Niv.Stoerung.St_4mA := FALSE;
   Zulauf_Niv.Stoerung.St_OF := FALSE;
   Zulauf_Niv.Stoerung.St_UF := FALSE;
   Zulauf_Niv.Stoerung.St_Kom_DP := FALSE;
   Zulauf_Niv.Stoerung.St_Kom_int := FALSE;
   Zulauf_Niv.Stoerung.St_int := FALSE;
   Zulauf_Niv.Stoerung.Res_7 := FALSE;
   Zulauf_Niv.Stoerung.GW_HH := FALSE;
   Zulauf_Niv.Stoerung.GW_H := FALSE;
   Zulauf_Niv.Stoerung.GW_L := FALSE;
   Zulauf_Niv.Stoerung.GW_LL := FALSE;
   Zulauf_Niv.Stoerung.Res_12 := FALSE;
   Zulauf_Niv.Stoerung.Res_13 := FALSE;
   Zulauf_Niv.Stoerung.Res_14 := FALSE;
   Zulauf_Niv.Stoerung.Res_15 := FALSE;
   Zulauf_Niv.Stoerung.Res_16 := FALSE;
   Zulauf_Niv.Stoerung.Res_17 := FALSE;
   Zulauf_Niv.Stoerung.Res_18 := FALSE;
   Zulauf_Niv.Stoerung.Res_19 := FALSE;
   Zulauf_Niv.Stoerung.Res_20 := FALSE;
   Zulauf_Niv.Stoerung.Res_21 := FALSE;
   Zulauf_Niv.Stoerung.Res_22 := FALSE;
   Zulauf_Niv.Stoerung.Res_23 := FALSE;
   Zulauf_Niv.Stoerung.Res_24 := FALSE;
   Zulauf_Niv.Stoerung.Res_25 := FALSE;
   Zulauf_Niv.Stoerung.Res_26 := FALSE;
   Zulauf_Niv.Stoerung.Res_27 := FALSE;
   Zulauf_Niv.Stoerung.Res_28 := FALSE;
   Zulauf_Niv.Stoerung.Res_29 := FALSE;
   Zulauf_Niv.Stoerung.Res_30 := FALSE;
   Zulauf_Niv.Stoerung.Res_31 := FALSE;
   Zulauf_Niv.MW_akt := 26.20959;
   Zulauf_DF.Status.BA_Nrm := TRUE;
   Zulauf_DF.Status.BA_Frz := FALSE;
   Zulauf_DF.Status.BA_EW := FALSE;
   Zulauf_DF.Status.BA_Sim := FALSE;
   Zulauf_DF.Status.BA_Wart := FALSE;
   Zulauf_DF.Status.Frg_HH := FALSE;
   Zulauf_DF.Status.Frg_H := FALSE;
   Zulauf_DF.Status.Frg_L := FALSE;
   Zulauf_DF.Status.Frg_LL := FALSE;
   Zulauf_DF.Status.SB_MW_frz := FALSE;
   Zulauf_DF.Status.SB_MW_EW := FALSE;
   Zulauf_DF.Status.BM_MW_ok := TRUE;
   Zulauf_DF.Status.BM_MW_frz := FALSE;
   Zulauf_DF.Status.BM_MW_EW := FALSE;
   Zulauf_DF.Status.BM_MW_Sim := FALSE;
   Zulauf_DF.Status.BM_MW_nok := FALSE;
   Zulauf_DF.Status.BM_MW_zw := FALSE;
   Zulauf_DF.Status.GW_Sp_H := FALSE;
   Zulauf_DF.Status.GW_Sp_L := FALSE;
   Zulauf_DF.Status.Res_19 := FALSE;
   Zulauf_DF.Status.Res_26 := FALSE;
   Zulauf_DF.Status.Res_27 := FALSE;
   Zulauf_DF.Status.Res_28 := FALSE;
   Zulauf_DF.Status.Res_29 := FALSE;
   Zulauf_DF.Status.Res_30 := FALSE;
   Zulauf_DF.Status.Res_31 := FALSE;
   Zulauf_DF.Status.Res_32 := FALSE;
   Zulauf_DF.Status.Res_33 := FALSE;
   Zulauf_DF.Status.Res_34 := FALSE;
   Zulauf_DF.Status.BB_AutoOk := TRUE;
   Zulauf_DF.Status.BB_SS := FALSE;
   Zulauf_DF.Status.BB_SSnq := FALSE;
   Zulauf_DF.Stoerung.St_allg := FALSE;
   Zulauf_DF.Stoerung.St_4mA := FALSE;
   Zulauf_DF.Stoerung.St_OF := FALSE;
   Zulauf_DF.Stoerung.St_UF := FALSE;
   Zulauf_DF.Stoerung.St_Kom_DP := FALSE;
   Zulauf_DF.Stoerung.St_Kom_int := FALSE;
   Zulauf_DF.Stoerung.St_int := FALSE;
   Zulauf_DF.Stoerung.Res_7 := FALSE;
   Zulauf_DF.Stoerung.GW_HH := FALSE;
   Zulauf_DF.Stoerung.GW_H := FALSE;
   Zulauf_DF.Stoerung.GW_L := FALSE;
   Zulauf_DF.Stoerung.GW_LL := FALSE;
   Zulauf_DF.Stoerung.Res_12 := FALSE;
   Zulauf_DF.Stoerung.Res_13 := FALSE;
   Zulauf_DF.Stoerung.Res_14 := FALSE;
   Zulauf_DF.Stoerung.Res_15 := FALSE;
   Zulauf_DF.Stoerung.Res_16 := FALSE;
   Zulauf_DF.Stoerung.Res_17 := FALSE;
   Zulauf_DF.Stoerung.Res_18 := FALSE;
   Zulauf_DF.Stoerung.Res_19 := FALSE;
   Zulauf_DF.Stoerung.Res_20 := FALSE;
   Zulauf_DF.Stoerung.Res_21 := FALSE;
   Zulauf_DF.Stoerung.Res_22 := FALSE;
   Zulauf_DF.Stoerung.Res_23 := FALSE;
   Zulauf_DF.Stoerung.Res_24 := FALSE;
   Zulauf_DF.Stoerung.Res_25 := FALSE;
   Zulauf_DF.Stoerung.Res_26 := FALSE;
   Zulauf_DF.Stoerung.Res_27 := FALSE;
   Zulauf_DF.Stoerung.Res_28 := FALSE;
   Zulauf_DF.Stoerung.Res_29 := FALSE;
   Zulauf_DF.Stoerung.Res_30 := FALSE;
   Zulauf_DF.Stoerung.Res_31 := FALSE;
   Zulauf_DF.MW_akt := 21.13387;
   Verteiler_pH.Status.BA_Nrm := TRUE;
   Verteiler_pH.Status.BA_Frz := FALSE;
   Verteiler_pH.Status.BA_EW := FALSE;
   Verteiler_pH.Status.BA_Sim := FALSE;
   Verteiler_pH.Status.BA_Wart := FALSE;
   Verteiler_pH.Status.Frg_HH := FALSE;
   Verteiler_pH.Status.Frg_H := FALSE;
   Verteiler_pH.Status.Frg_L := FALSE;
   Verteiler_pH.Status.Frg_LL := FALSE;
   Verteiler_pH.Status.SB_MW_frz := FALSE;
   Verteiler_pH.Status.SB_MW_EW := FALSE;
   Verteiler_pH.Status.BM_MW_ok := TRUE;
   Verteiler_pH.Status.BM_MW_frz := FALSE;
   Verteiler_pH.Status.BM_MW_EW := FALSE;
   Verteiler_pH.Status.BM_MW_Sim := FALSE;
   Verteiler_pH.Status.BM_MW_nok := FALSE;
   Verteiler_pH.Status.BM_MW_zw := FALSE;
   Verteiler_pH.Status.GW_Sp_H := FALSE;
   Verteiler_pH.Status.GW_Sp_L := FALSE;
   Verteiler_pH.Status.Res_19 := FALSE;
   Verteiler_pH.Status.Res_26 := FALSE;
   Verteiler_pH.Status.Res_27 := FALSE;
   Verteiler_pH.Status.Res_28 := FALSE;
   Verteiler_pH.Status.Res_29 := FALSE;
   Verteiler_pH.Status.Res_30 := FALSE;
   Verteiler_pH.Status.Res_31 := FALSE;
   Verteiler_pH.Status.Res_32 := FALSE;
   Verteiler_pH.Status.Res_33 := FALSE;
   Verteiler_pH.Status.Res_34 := FALSE;
   Verteiler_pH.Status.BB_AutoOk := TRUE;
   Verteiler_pH.Status.BB_SS := FALSE;
   Verteiler_pH.Status.BB_SSnq := FALSE;
   Verteiler_pH.Stoerung.St_allg := FALSE;
   Verteiler_pH.Stoerung.St_4mA := FALSE;
   Verteiler_pH.Stoerung.St_OF := FALSE;
   Verteiler_pH.Stoerung.St_UF := FALSE;
   Verteiler_pH.Stoerung.St_Kom_DP := FALSE;
   Verteiler_pH.Stoerung.St_Kom_int := FALSE;
   Verteiler_pH.Stoerung.St_int := FALSE;
   Verteiler_pH.Stoerung.Res_7 := FALSE;
   Verteiler_pH.Stoerung.GW_HH := FALSE;
   Verteiler_pH.Stoerung.GW_H := FALSE;
   Verteiler_pH.Stoerung.GW_L := FALSE;
   Verteiler_pH.Stoerung.GW_LL := FALSE;
   Verteiler_pH.Stoerung.Res_12 := FALSE;
   Verteiler_pH.Stoerung.Res_13 := FALSE;
   Verteiler_pH.Stoerung.Res_14 := FALSE;
   Verteiler_pH.Stoerung.Res_15 := FALSE;
   Verteiler_pH.Stoerung.Res_16 := FALSE;
   Verteiler_pH.Stoerung.Res_17 := FALSE;
   Verteiler_pH.Stoerung.Res_18 := FALSE;
   Verteiler_pH.Stoerung.Res_19 := FALSE;
   Verteiler_pH.Stoerung.Res_20 := FALSE;
   Verteiler_pH.Stoerung.Res_21 := FALSE;
   Verteiler_pH.Stoerung.Res_22 := FALSE;
   Verteiler_pH.Stoerung.Res_23 := FALSE;
   Verteiler_pH.Stoerung.Res_24 := FALSE;
   Verteiler_pH.Stoerung.Res_25 := FALSE;
   Verteiler_pH.Stoerung.Res_26 := FALSE;
   Verteiler_pH.Stoerung.Res_27 := FALSE;
   Verteiler_pH.Stoerung.Res_28 := FALSE;
   Verteiler_pH.Stoerung.Res_29 := FALSE;
   Verteiler_pH.Stoerung.Res_30 := FALSE;
   Verteiler_pH.Stoerung.Res_31 := FALSE;
   Verteiler_pH.MW_akt := 2.0;
   Verteiler_O2.Status.BA_Nrm := TRUE;
   Verteiler_O2.Status.BA_Frz := FALSE;
   Verteiler_O2.Status.BA_EW := FALSE;
   Verteiler_O2.Status.BA_Sim := FALSE;
   Verteiler_O2.Status.BA_Wart := FALSE;
   Verteiler_O2.Status.Frg_HH := FALSE;
   Verteiler_O2.Status.Frg_H := FALSE;
   Verteiler_O2.Status.Frg_L := FALSE;
   Verteiler_O2.Status.Frg_LL := FALSE;
   Verteiler_O2.Status.SB_MW_frz := FALSE;
   Verteiler_O2.Status.SB_MW_EW := FALSE;
   Verteiler_O2.Status.BM_MW_ok := TRUE;
   Verteiler_O2.Status.BM_MW_frz := FALSE;
   Verteiler_O2.Status.BM_MW_EW := FALSE;
   Verteiler_O2.Status.BM_MW_Sim := FALSE;
   Verteiler_O2.Status.BM_MW_nok := FALSE;
   Verteiler_O2.Status.BM_MW_zw := FALSE;
   Verteiler_O2.Status.GW_Sp_H := FALSE;
   Verteiler_O2.Status.GW_Sp_L := FALSE;
   Verteiler_O2.Status.Res_19 := FALSE;
   Verteiler_O2.Status.Res_26 := FALSE;
   Verteiler_O2.Status.Res_27 := FALSE;
   Verteiler_O2.Status.Res_28 := FALSE;
   Verteiler_O2.Status.Res_29 := FALSE;
   Verteiler_O2.Status.Res_30 := FALSE;
   Verteiler_O2.Status.Res_31 := FALSE;
   Verteiler_O2.Status.Res_32 := FALSE;
   Verteiler_O2.Status.Res_33 := FALSE;
   Verteiler_O2.Status.Res_34 := FALSE;
   Verteiler_O2.Status.BB_AutoOk := TRUE;
   Verteiler_O2.Status.BB_SS := FALSE;
   Verteiler_O2.Status.BB_SSnq := FALSE;
   Verteiler_O2.Stoerung.St_allg := FALSE;
   Verteiler_O2.Stoerung.St_4mA := FALSE;
   Verteiler_O2.Stoerung.St_OF := FALSE;
   Verteiler_O2.Stoerung.St_UF := FALSE;
   Verteiler_O2.Stoerung.St_Kom_DP := FALSE;
   Verteiler_O2.Stoerung.St_Kom_int := FALSE;
   Verteiler_O2.Stoerung.St_int := FALSE;
   Verteiler_O2.Stoerung.Res_7 := FALSE;
   Verteiler_O2.Stoerung.GW_HH := FALSE;
   Verteiler_O2.Stoerung.GW_H := FALSE;
   Verteiler_O2.Stoerung.GW_L := FALSE;
   Verteiler_O2.Stoerung.GW_LL := FALSE;
   Verteiler_O2.Stoerung.Res_12 := FALSE;
   Verteiler_O2.Stoerung.Res_13 := FALSE;
   Verteiler_O2.Stoerung.Res_14 := FALSE;
   Verteiler_O2.Stoerung.Res_15 := FALSE;
   Verteiler_O2.Stoerung.Res_16 := FALSE;
   Verteiler_O2.Stoerung.Res_17 := FALSE;
   Verteiler_O2.Stoerung.Res_18 := FALSE;
   Verteiler_O2.Stoerung.Res_19 := FALSE;
   Verteiler_O2.Stoerung.Res_20 := FALSE;
   Verteiler_O2.Stoerung.Res_21 := FALSE;
   Verteiler_O2.Stoerung.Res_22 := FALSE;
   Verteiler_O2.Stoerung.Res_23 := FALSE;
   Verteiler_O2.Stoerung.Res_24 := FALSE;
   Verteiler_O2.Stoerung.Res_25 := FALSE;
   Verteiler_O2.Stoerung.Res_26 := FALSE;
   Verteiler_O2.Stoerung.Res_27 := FALSE;
   Verteiler_O2.Stoerung.Res_28 := FALSE;
   Verteiler_O2.Stoerung.Res_29 := FALSE;
   Verteiler_O2.Stoerung.Res_30 := FALSE;
   Verteiler_O2.Stoerung.Res_31 := FALSE;
   Verteiler_O2.MW_akt := 0.0;
   Verteiler_Temp.Status.BA_Nrm := TRUE;
   Verteiler_Temp.Status.BA_Frz := FALSE;
   Verteiler_Temp.Status.BA_EW := FALSE;
   Verteiler_Temp.Status.BA_Sim := FALSE;
   Verteiler_Temp.Status.BA_Wart := FALSE;
   Verteiler_Temp.Status.Frg_HH := FALSE;
   Verteiler_Temp.Status.Frg_H := FALSE;
   Verteiler_Temp.Status.Frg_L := FALSE;
   Verteiler_Temp.Status.Frg_LL := FALSE;
   Verteiler_Temp.Status.SB_MW_frz := FALSE;
   Verteiler_Temp.Status.SB_MW_EW := FALSE;
   Verteiler_Temp.Status.BM_MW_ok := TRUE;
   Verteiler_Temp.Status.BM_MW_frz := FALSE;
   Verteiler_Temp.Status.BM_MW_EW := FALSE;
   Verteiler_Temp.Status.BM_MW_Sim := FALSE;
   Verteiler_Temp.Status.BM_MW_nok := FALSE;
   Verteiler_Temp.Status.BM_MW_zw := FALSE;
   Verteiler_Temp.Status.GW_Sp_H := FALSE;
   Verteiler_Temp.Status.GW_Sp_L := FALSE;
   Verteiler_Temp.Status.Res_19 := FALSE;
   Verteiler_Temp.Status.Res_26 := FALSE;
   Verteiler_Temp.Status.Res_27 := FALSE;
   Verteiler_Temp.Status.Res_28 := FALSE;
   Verteiler_Temp.Status.Res_29 := FALSE;
   Verteiler_Temp.Status.Res_30 := FALSE;
   Verteiler_Temp.Status.Res_31 := FALSE;
   Verteiler_Temp.Status.Res_32 := FALSE;
   Verteiler_Temp.Status.Res_33 := FALSE;
   Verteiler_Temp.Status.Res_34 := FALSE;
   Verteiler_Temp.Status.BB_AutoOk := TRUE;
   Verteiler_Temp.Status.BB_SS := FALSE;
   Verteiler_Temp.Status.BB_SSnq := FALSE;
   Verteiler_Temp.Stoerung.St_allg := FALSE;
   Verteiler_Temp.Stoerung.St_4mA := FALSE;
   Verteiler_Temp.Stoerung.St_OF := FALSE;
   Verteiler_Temp.Stoerung.St_UF := FALSE;
   Verteiler_Temp.Stoerung.St_Kom_DP := FALSE;
   Verteiler_Temp.Stoerung.St_Kom_int := FALSE;
   Verteiler_Temp.Stoerung.St_int := FALSE;
   Verteiler_Temp.Stoerung.Res_7 := FALSE;
   Verteiler_Temp.Stoerung.GW_HH := FALSE;
   Verteiler_Temp.Stoerung.GW_H := FALSE;
   Verteiler_Temp.Stoerung.GW_L := FALSE;
   Verteiler_Temp.Stoerung.GW_LL := FALSE;
   Verteiler_Temp.Stoerung.Res_12 := FALSE;
   Verteiler_Temp.Stoerung.Res_13 := FALSE;
   Verteiler_Temp.Stoerung.Res_14 := FALSE;
   Verteiler_Temp.Stoerung.Res_15 := FALSE;
   Verteiler_Temp.Stoerung.Res_16 := FALSE;
   Verteiler_Temp.Stoerung.Res_17 := FALSE;
   Verteiler_Temp.Stoerung.Res_18 := FALSE;
   Verteiler_Temp.Stoerung.Res_19 := FALSE;
   Verteiler_Temp.Stoerung.Res_20 := FALSE;
   Verteiler_Temp.Stoerung.Res_21 := FALSE;
   Verteiler_Temp.Stoerung.Res_22 := FALSE;
   Verteiler_Temp.Stoerung.Res_23 := FALSE;
   Verteiler_Temp.Stoerung.Res_24 := FALSE;
   Verteiler_Temp.Stoerung.Res_25 := FALSE;
   Verteiler_Temp.Stoerung.Res_26 := FALSE;
   Verteiler_Temp.Stoerung.Res_27 := FALSE;
   Verteiler_Temp.Stoerung.Res_28 := FALSE;
   Verteiler_Temp.Stoerung.Res_29 := FALSE;
   Verteiler_Temp.Stoerung.Res_30 := FALSE;
   Verteiler_Temp.Stoerung.Res_31 := FALSE;
   Verteiler_Temp.MW_akt := 0.0;
   BB_UeSS_DF.Status.BA_Nrm := TRUE;
   BB_UeSS_DF.Status.BA_Frz := FALSE;
   BB_UeSS_DF.Status.BA_EW := FALSE;
   BB_UeSS_DF.Status.BA_Sim := FALSE;
   BB_UeSS_DF.Status.BA_Wart := FALSE;
   BB_UeSS_DF.Status.Frg_HH := FALSE;
   BB_UeSS_DF.Status.Frg_H := FALSE;
   BB_UeSS_DF.Status.Frg_L := FALSE;
   BB_UeSS_DF.Status.Frg_LL := FALSE;
   BB_UeSS_DF.Status.SB_MW_frz := FALSE;
   BB_UeSS_DF.Status.SB_MW_EW := FALSE;
   BB_UeSS_DF.Status.BM_MW_ok := TRUE;
   BB_UeSS_DF.Status.BM_MW_frz := FALSE;
   BB_UeSS_DF.Status.BM_MW_EW := FALSE;
   BB_UeSS_DF.Status.BM_MW_Sim := FALSE;
   BB_UeSS_DF.Status.BM_MW_nok := FALSE;
   BB_UeSS_DF.Status.BM_MW_zw := FALSE;
   BB_UeSS_DF.Status.GW_Sp_H := FALSE;
   BB_UeSS_DF.Status.GW_Sp_L := FALSE;
   BB_UeSS_DF.Status.Res_19 := FALSE;
   BB_UeSS_DF.Status.Res_26 := FALSE;
   BB_UeSS_DF.Status.Res_27 := FALSE;
   BB_UeSS_DF.Status.Res_28 := FALSE;
   BB_UeSS_DF.Status.Res_29 := FALSE;
   BB_UeSS_DF.Status.Res_30 := FALSE;
   BB_UeSS_DF.Status.Res_31 := FALSE;
   BB_UeSS_DF.Status.Res_32 := FALSE;
   BB_UeSS_DF.Status.Res_33 := FALSE;
   BB_UeSS_DF.Status.Res_34 := FALSE;
   BB_UeSS_DF.Status.BB_AutoOk := TRUE;
   BB_UeSS_DF.Status.BB_SS := FALSE;
   BB_UeSS_DF.Status.BB_SSnq := FALSE;
   BB_UeSS_DF.Stoerung.St_allg := FALSE;
   BB_UeSS_DF.Stoerung.St_4mA := FALSE;
   BB_UeSS_DF.Stoerung.St_OF := FALSE;
   BB_UeSS_DF.Stoerung.St_UF := FALSE;
   BB_UeSS_DF.Stoerung.St_Kom_DP := FALSE;
   BB_UeSS_DF.Stoerung.St_Kom_int := FALSE;
   BB_UeSS_DF.Stoerung.St_int := FALSE;
   BB_UeSS_DF.Stoerung.Res_7 := FALSE;
   BB_UeSS_DF.Stoerung.GW_HH := FALSE;
   BB_UeSS_DF.Stoerung.GW_H := FALSE;
   BB_UeSS_DF.Stoerung.GW_L := FALSE;
   BB_UeSS_DF.Stoerung.GW_LL := FALSE;
   BB_UeSS_DF.Stoerung.Res_12 := FALSE;
   BB_UeSS_DF.Stoerung.Res_13 := FALSE;
   BB_UeSS_DF.Stoerung.Res_14 := FALSE;
   BB_UeSS_DF.Stoerung.Res_15 := FALSE;
   BB_UeSS_DF.Stoerung.Res_16 := FALSE;
   BB_UeSS_DF.Stoerung.Res_17 := FALSE;
   BB_UeSS_DF.Stoerung.Res_18 := FALSE;
   BB_UeSS_DF.Stoerung.Res_19 := FALSE;
   BB_UeSS_DF.Stoerung.Res_20 := FALSE;
   BB_UeSS_DF.Stoerung.Res_21 := FALSE;
   BB_UeSS_DF.Stoerung.Res_22 := FALSE;
   BB_UeSS_DF.Stoerung.Res_23 := FALSE;
   BB_UeSS_DF.Stoerung.Res_24 := FALSE;
   BB_UeSS_DF.Stoerung.Res_25 := FALSE;
   BB_UeSS_DF.Stoerung.Res_26 := FALSE;
   BB_UeSS_DF.Stoerung.Res_27 := FALSE;
   BB_UeSS_DF.Stoerung.Res_28 := FALSE;
   BB_UeSS_DF.Stoerung.Res_29 := FALSE;
   BB_UeSS_DF.Stoerung.Res_30 := FALSE;
   BB_UeSS_DF.Stoerung.Res_31 := FALSE;
   BB_UeSS_DF.MW_akt := -0.0067815;
   Ablauf_DF.Status.BA_Nrm := TRUE;
   Ablauf_DF.Status.BA_Frz := FALSE;
   Ablauf_DF.Status.BA_EW := FALSE;
   Ablauf_DF.Status.BA_Sim := FALSE;
   Ablauf_DF.Status.BA_Wart := FALSE;
   Ablauf_DF.Status.Frg_HH := FALSE;
   Ablauf_DF.Status.Frg_H := FALSE;
   Ablauf_DF.Status.Frg_L := FALSE;
   Ablauf_DF.Status.Frg_LL := FALSE;
   Ablauf_DF.Status.SB_MW_frz := FALSE;
   Ablauf_DF.Status.SB_MW_EW := FALSE;
   Ablauf_DF.Status.BM_MW_ok := TRUE;
   Ablauf_DF.Status.BM_MW_frz := FALSE;
   Ablauf_DF.Status.BM_MW_EW := FALSE;
   Ablauf_DF.Status.BM_MW_Sim := FALSE;
   Ablauf_DF.Status.BM_MW_nok := FALSE;
   Ablauf_DF.Status.BM_MW_zw := FALSE;
   Ablauf_DF.Status.GW_Sp_H := FALSE;
   Ablauf_DF.Status.GW_Sp_L := FALSE;
   Ablauf_DF.Status.Res_19 := FALSE;
   Ablauf_DF.Status.Res_26 := FALSE;
   Ablauf_DF.Status.Res_27 := FALSE;
   Ablauf_DF.Status.Res_28 := FALSE;
   Ablauf_DF.Status.Res_29 := FALSE;
   Ablauf_DF.Status.Res_30 := FALSE;
   Ablauf_DF.Status.Res_31 := FALSE;
   Ablauf_DF.Status.Res_32 := FALSE;
   Ablauf_DF.Status.Res_33 := FALSE;
   Ablauf_DF.Status.Res_34 := FALSE;
   Ablauf_DF.Status.BB_AutoOk := TRUE;
   Ablauf_DF.Status.BB_SS := FALSE;
   Ablauf_DF.Status.BB_SSnq := FALSE;
   Ablauf_DF.Stoerung.St_allg := FALSE;
   Ablauf_DF.Stoerung.St_4mA := FALSE;
   Ablauf_DF.Stoerung.St_OF := FALSE;
   Ablauf_DF.Stoerung.St_UF := FALSE;
   Ablauf_DF.Stoerung.St_Kom_DP := FALSE;
   Ablauf_DF.Stoerung.St_Kom_int := FALSE;
   Ablauf_DF.Stoerung.St_int := FALSE;
   Ablauf_DF.Stoerung.Res_7 := FALSE;
   Ablauf_DF.Stoerung.GW_HH := FALSE;
   Ablauf_DF.Stoerung.GW_H := FALSE;
   Ablauf_DF.Stoerung.GW_L := FALSE;
   Ablauf_DF.Stoerung.GW_LL := FALSE;
   Ablauf_DF.Stoerung.Res_12 := FALSE;
   Ablauf_DF.Stoerung.Res_13 := FALSE;
   Ablauf_DF.Stoerung.Res_14 := FALSE;
   Ablauf_DF.Stoerung.Res_15 := FALSE;
   Ablauf_DF.Stoerung.Res_16 := FALSE;
   Ablauf_DF.Stoerung.Res_17 := FALSE;
   Ablauf_DF.Stoerung.Res_18 := FALSE;
   Ablauf_DF.Stoerung.Res_19 := FALSE;
   Ablauf_DF.Stoerung.Res_20 := FALSE;
   Ablauf_DF.Stoerung.Res_21 := FALSE;
   Ablauf_DF.Stoerung.Res_22 := FALSE;
   Ablauf_DF.Stoerung.Res_23 := FALSE;
   Ablauf_DF.Stoerung.Res_24 := FALSE;
   Ablauf_DF.Stoerung.Res_25 := FALSE;
   Ablauf_DF.Stoerung.Res_26 := FALSE;
   Ablauf_DF.Stoerung.Res_27 := FALSE;
   Ablauf_DF.Stoerung.Res_28 := FALSE;
   Ablauf_DF.Stoerung.Res_29 := FALSE;
   Ablauf_DF.Stoerung.Res_30 := FALSE;
   Ablauf_DF.Stoerung.Res_31 := FALSE;
   Ablauf_DF.MW_akt := 11.20182;
   Ablauf_pH.Status.BA_Nrm := TRUE;
   Ablauf_pH.Status.BA_Frz := FALSE;
   Ablauf_pH.Status.BA_EW := FALSE;
   Ablauf_pH.Status.BA_Sim := FALSE;
   Ablauf_pH.Status.BA_Wart := FALSE;
   Ablauf_pH.Status.Frg_HH := FALSE;
   Ablauf_pH.Status.Frg_H := FALSE;
   Ablauf_pH.Status.Frg_L := FALSE;
   Ablauf_pH.Status.Frg_LL := FALSE;
   Ablauf_pH.Status.SB_MW_frz := FALSE;
   Ablauf_pH.Status.SB_MW_EW := FALSE;
   Ablauf_pH.Status.BM_MW_ok := TRUE;
   Ablauf_pH.Status.BM_MW_frz := FALSE;
   Ablauf_pH.Status.BM_MW_EW := FALSE;
   Ablauf_pH.Status.BM_MW_Sim := FALSE;
   Ablauf_pH.Status.BM_MW_nok := FALSE;
   Ablauf_pH.Status.BM_MW_zw := FALSE;
   Ablauf_pH.Status.GW_Sp_H := FALSE;
   Ablauf_pH.Status.GW_Sp_L := FALSE;
   Ablauf_pH.Status.Res_19 := FALSE;
   Ablauf_pH.Status.Res_26 := FALSE;
   Ablauf_pH.Status.Res_27 := FALSE;
   Ablauf_pH.Status.Res_28 := FALSE;
   Ablauf_pH.Status.Res_29 := FALSE;
   Ablauf_pH.Status.Res_30 := FALSE;
   Ablauf_pH.Status.Res_31 := FALSE;
   Ablauf_pH.Status.Res_32 := FALSE;
   Ablauf_pH.Status.Res_33 := FALSE;
   Ablauf_pH.Status.Res_34 := FALSE;
   Ablauf_pH.Status.BB_AutoOk := TRUE;
   Ablauf_pH.Status.BB_SS := FALSE;
   Ablauf_pH.Status.BB_SSnq := FALSE;
   Ablauf_pH.Stoerung.St_allg := FALSE;
   Ablauf_pH.Stoerung.St_4mA := FALSE;
   Ablauf_pH.Stoerung.St_OF := FALSE;
   Ablauf_pH.Stoerung.St_UF := FALSE;
   Ablauf_pH.Stoerung.St_Kom_DP := FALSE;
   Ablauf_pH.Stoerung.St_Kom_int := FALSE;
   Ablauf_pH.Stoerung.St_int := FALSE;
   Ablauf_pH.Stoerung.Res_7 := FALSE;
   Ablauf_pH.Stoerung.GW_HH := FALSE;
   Ablauf_pH.Stoerung.GW_H := FALSE;
   Ablauf_pH.Stoerung.GW_L := FALSE;
   Ablauf_pH.Stoerung.GW_LL := FALSE;
   Ablauf_pH.Stoerung.Res_12 := FALSE;
   Ablauf_pH.Stoerung.Res_13 := FALSE;
   Ablauf_pH.Stoerung.Res_14 := FALSE;
   Ablauf_pH.Stoerung.Res_15 := FALSE;
   Ablauf_pH.Stoerung.Res_16 := FALSE;
   Ablauf_pH.Stoerung.Res_17 := FALSE;
   Ablauf_pH.Stoerung.Res_18 := FALSE;
   Ablauf_pH.Stoerung.Res_19 := FALSE;
   Ablauf_pH.Stoerung.Res_20 := FALSE;
   Ablauf_pH.Stoerung.Res_21 := FALSE;
   Ablauf_pH.Stoerung.Res_22 := FALSE;
   Ablauf_pH.Stoerung.Res_23 := FALSE;
   Ablauf_pH.Stoerung.Res_24 := FALSE;
   Ablauf_pH.Stoerung.Res_25 := FALSE;
   Ablauf_pH.Stoerung.Res_26 := FALSE;
   Ablauf_pH.Stoerung.Res_27 := FALSE;
   Ablauf_pH.Stoerung.Res_28 := FALSE;
   Ablauf_pH.Stoerung.Res_29 := FALSE;
   Ablauf_pH.Stoerung.Res_30 := FALSE;
   Ablauf_pH.Stoerung.Res_31 := FALSE;
   Ablauf_pH.MW_akt := 7.054876;
   Ablauf_O2.Status.BA_Nrm := TRUE;
   Ablauf_O2.Status.BA_Frz := FALSE;
   Ablauf_O2.Status.BA_EW := FALSE;
   Ablauf_O2.Status.BA_Sim := FALSE;
   Ablauf_O2.Status.BA_Wart := FALSE;
   Ablauf_O2.Status.Frg_HH := FALSE;
   Ablauf_O2.Status.Frg_H := FALSE;
   Ablauf_O2.Status.Frg_L := FALSE;
   Ablauf_O2.Status.Frg_LL := FALSE;
   Ablauf_O2.Status.SB_MW_frz := FALSE;
   Ablauf_O2.Status.SB_MW_EW := FALSE;
   Ablauf_O2.Status.BM_MW_ok := TRUE;
   Ablauf_O2.Status.BM_MW_frz := FALSE;
   Ablauf_O2.Status.BM_MW_EW := FALSE;
   Ablauf_O2.Status.BM_MW_Sim := FALSE;
   Ablauf_O2.Status.BM_MW_nok := FALSE;
   Ablauf_O2.Status.BM_MW_zw := FALSE;
   Ablauf_O2.Status.GW_Sp_H := FALSE;
   Ablauf_O2.Status.GW_Sp_L := FALSE;
   Ablauf_O2.Status.Res_19 := FALSE;
   Ablauf_O2.Status.Res_26 := FALSE;
   Ablauf_O2.Status.Res_27 := FALSE;
   Ablauf_O2.Status.Res_28 := FALSE;
   Ablauf_O2.Status.Res_29 := FALSE;
   Ablauf_O2.Status.Res_30 := FALSE;
   Ablauf_O2.Status.Res_31 := FALSE;
   Ablauf_O2.Status.Res_32 := FALSE;
   Ablauf_O2.Status.Res_33 := FALSE;
   Ablauf_O2.Status.Res_34 := FALSE;
   Ablauf_O2.Status.BB_AutoOk := TRUE;
   Ablauf_O2.Status.BB_SS := FALSE;
   Ablauf_O2.Status.BB_SSnq := FALSE;
   Ablauf_O2.Stoerung.St_allg := FALSE;
   Ablauf_O2.Stoerung.St_4mA := FALSE;
   Ablauf_O2.Stoerung.St_OF := FALSE;
   Ablauf_O2.Stoerung.St_UF := FALSE;
   Ablauf_O2.Stoerung.St_Kom_DP := FALSE;
   Ablauf_O2.Stoerung.St_Kom_int := FALSE;
   Ablauf_O2.Stoerung.St_int := FALSE;
   Ablauf_O2.Stoerung.Res_7 := FALSE;
   Ablauf_O2.Stoerung.GW_HH := FALSE;
   Ablauf_O2.Stoerung.GW_H := FALSE;
   Ablauf_O2.Stoerung.GW_L := FALSE;
   Ablauf_O2.Stoerung.GW_LL := FALSE;
   Ablauf_O2.Stoerung.Res_12 := FALSE;
   Ablauf_O2.Stoerung.Res_13 := FALSE;
   Ablauf_O2.Stoerung.Res_14 := FALSE;
   Ablauf_O2.Stoerung.Res_15 := FALSE;
   Ablauf_O2.Stoerung.Res_16 := FALSE;
   Ablauf_O2.Stoerung.Res_17 := FALSE;
   Ablauf_O2.Stoerung.Res_18 := FALSE;
   Ablauf_O2.Stoerung.Res_19 := FALSE;
   Ablauf_O2.Stoerung.Res_20 := FALSE;
   Ablauf_O2.Stoerung.Res_21 := FALSE;
   Ablauf_O2.Stoerung.Res_22 := FALSE;
   Ablauf_O2.Stoerung.Res_23 := FALSE;
   Ablauf_O2.Stoerung.Res_24 := FALSE;
   Ablauf_O2.Stoerung.Res_25 := FALSE;
   Ablauf_O2.Stoerung.Res_26 := FALSE;
   Ablauf_O2.Stoerung.Res_27 := FALSE;
   Ablauf_O2.Stoerung.Res_28 := FALSE;
   Ablauf_O2.Stoerung.Res_29 := FALSE;
   Ablauf_O2.Stoerung.Res_30 := FALSE;
   Ablauf_O2.Stoerung.Res_31 := FALSE;
   Ablauf_O2.MW_akt := 1.478322;
   Ablauf_Temp.Status.BA_Nrm := TRUE;
   Ablauf_Temp.Status.BA_Frz := FALSE;
   Ablauf_Temp.Status.BA_EW := FALSE;
   Ablauf_Temp.Status.BA_Sim := FALSE;
   Ablauf_Temp.Status.BA_Wart := FALSE;
   Ablauf_Temp.Status.Frg_HH := FALSE;
   Ablauf_Temp.Status.Frg_H := FALSE;
   Ablauf_Temp.Status.Frg_L := FALSE;
   Ablauf_Temp.Status.Frg_LL := FALSE;
   Ablauf_Temp.Status.SB_MW_frz := FALSE;
   Ablauf_Temp.Status.SB_MW_EW := FALSE;
   Ablauf_Temp.Status.BM_MW_ok := TRUE;
   Ablauf_Temp.Status.BM_MW_frz := FALSE;
   Ablauf_Temp.Status.BM_MW_EW := FALSE;
   Ablauf_Temp.Status.BM_MW_Sim := FALSE;
   Ablauf_Temp.Status.BM_MW_nok := FALSE;
   Ablauf_Temp.Status.BM_MW_zw := FALSE;
   Ablauf_Temp.Status.GW_Sp_H := FALSE;
   Ablauf_Temp.Status.GW_Sp_L := FALSE;
   Ablauf_Temp.Status.Res_19 := FALSE;
   Ablauf_Temp.Status.Res_26 := FALSE;
   Ablauf_Temp.Status.Res_27 := FALSE;
   Ablauf_Temp.Status.Res_28 := FALSE;
   Ablauf_Temp.Status.Res_29 := FALSE;
   Ablauf_Temp.Status.Res_30 := FALSE;
   Ablauf_Temp.Status.Res_31 := FALSE;
   Ablauf_Temp.Status.Res_32 := FALSE;
   Ablauf_Temp.Status.Res_33 := FALSE;
   Ablauf_Temp.Status.Res_34 := FALSE;
   Ablauf_Temp.Status.BB_AutoOk := TRUE;
   Ablauf_Temp.Status.BB_SS := FALSE;
   Ablauf_Temp.Status.BB_SSnq := FALSE;
   Ablauf_Temp.Stoerung.St_allg := FALSE;
   Ablauf_Temp.Stoerung.St_4mA := FALSE;
   Ablauf_Temp.Stoerung.St_OF := FALSE;
   Ablauf_Temp.Stoerung.St_UF := FALSE;
   Ablauf_Temp.Stoerung.St_Kom_DP := FALSE;
   Ablauf_Temp.Stoerung.St_Kom_int := FALSE;
   Ablauf_Temp.Stoerung.St_int := FALSE;
   Ablauf_Temp.Stoerung.Res_7 := FALSE;
   Ablauf_Temp.Stoerung.GW_HH := FALSE;
   Ablauf_Temp.Stoerung.GW_H := FALSE;
   Ablauf_Temp.Stoerung.GW_L := FALSE;
   Ablauf_Temp.Stoerung.GW_LL := FALSE;
   Ablauf_Temp.Stoerung.Res_12 := FALSE;
   Ablauf_Temp.Stoerung.Res_13 := FALSE;
   Ablauf_Temp.Stoerung.Res_14 := FALSE;
   Ablauf_Temp.Stoerung.Res_15 := FALSE;
   Ablauf_Temp.Stoerung.Res_16 := FALSE;
   Ablauf_Temp.Stoerung.Res_17 := FALSE;
   Ablauf_Temp.Stoerung.Res_18 := FALSE;
   Ablauf_Temp.Stoerung.Res_19 := FALSE;
   Ablauf_Temp.Stoerung.Res_20 := FALSE;
   Ablauf_Temp.Stoerung.Res_21 := FALSE;
   Ablauf_Temp.Stoerung.Res_22 := FALSE;
   Ablauf_Temp.Stoerung.Res_23 := FALSE;
   Ablauf_Temp.Stoerung.Res_24 := FALSE;
   Ablauf_Temp.Stoerung.Res_25 := FALSE;
   Ablauf_Temp.Stoerung.Res_26 := FALSE;
   Ablauf_Temp.Stoerung.Res_27 := FALSE;
   Ablauf_Temp.Stoerung.Res_28 := FALSE;
   Ablauf_Temp.Stoerung.Res_29 := FALSE;
   Ablauf_Temp.Stoerung.Res_30 := FALSE;
   Ablauf_Temp.Stoerung.Res_31 := FALSE;
   Ablauf_Temp.MW_akt := 12.91898;
   Schlamm_ED_Niv.Status.BA_Nrm := TRUE;
   Schlamm_ED_Niv.Status.BA_Frz := FALSE;
   Schlamm_ED_Niv.Status.BA_EW := FALSE;
   Schlamm_ED_Niv.Status.BA_Sim := FALSE;
   Schlamm_ED_Niv.Status.BA_Wart := FALSE;
   Schlamm_ED_Niv.Status.Frg_HH := FALSE;
   Schlamm_ED_Niv.Status.Frg_H := FALSE;
   Schlamm_ED_Niv.Status.Frg_L := FALSE;
   Schlamm_ED_Niv.Status.Frg_LL := FALSE;
   Schlamm_ED_Niv.Status.SB_MW_frz := FALSE;
   Schlamm_ED_Niv.Status.SB_MW_EW := FALSE;
   Schlamm_ED_Niv.Status.BM_MW_ok := TRUE;
   Schlamm_ED_Niv.Status.BM_MW_frz := FALSE;
   Schlamm_ED_Niv.Status.BM_MW_EW := FALSE;
   Schlamm_ED_Niv.Status.BM_MW_Sim := FALSE;
   Schlamm_ED_Niv.Status.BM_MW_nok := FALSE;
   Schlamm_ED_Niv.Status.BM_MW_zw := FALSE;
   Schlamm_ED_Niv.Status.GW_Sp_H := FALSE;
   Schlamm_ED_Niv.Status.GW_Sp_L := FALSE;
   Schlamm_ED_Niv.Status.Res_19 := FALSE;
   Schlamm_ED_Niv.Status.Res_26 := FALSE;
   Schlamm_ED_Niv.Status.Res_27 := FALSE;
   Schlamm_ED_Niv.Status.Res_28 := FALSE;
   Schlamm_ED_Niv.Status.Res_29 := FALSE;
   Schlamm_ED_Niv.Status.Res_30 := FALSE;
   Schlamm_ED_Niv.Status.Res_31 := FALSE;
   Schlamm_ED_Niv.Status.Res_32 := FALSE;
   Schlamm_ED_Niv.Status.Res_33 := FALSE;
   Schlamm_ED_Niv.Status.Res_34 := FALSE;
   Schlamm_ED_Niv.Status.BB_AutoOk := TRUE;
   Schlamm_ED_Niv.Status.BB_SS := FALSE;
   Schlamm_ED_Niv.Status.BB_SSnq := FALSE;
   Schlamm_ED_Niv.Stoerung.St_allg := FALSE;
   Schlamm_ED_Niv.Stoerung.St_4mA := FALSE;
   Schlamm_ED_Niv.Stoerung.St_OF := FALSE;
   Schlamm_ED_Niv.Stoerung.St_UF := FALSE;
   Schlamm_ED_Niv.Stoerung.St_Kom_DP := FALSE;
   Schlamm_ED_Niv.Stoerung.St_Kom_int := FALSE;
   Schlamm_ED_Niv.Stoerung.St_int := FALSE;
   Schlamm_ED_Niv.Stoerung.Res_7 := FALSE;
   Schlamm_ED_Niv.Stoerung.GW_HH := FALSE;
   Schlamm_ED_Niv.Stoerung.GW_H := FALSE;
   Schlamm_ED_Niv.Stoerung.GW_L := FALSE;
   Schlamm_ED_Niv.Stoerung.GW_LL := FALSE;
   Schlamm_ED_Niv.Stoerung.Res_12 := FALSE;
   Schlamm_ED_Niv.Stoerung.Res_13 := FALSE;
   Schlamm_ED_Niv.Stoerung.Res_14 := FALSE;
   Schlamm_ED_Niv.Stoerung.Res_15 := FALSE;
   Schlamm_ED_Niv.Stoerung.Res_16 := FALSE;
   Schlamm_ED_Niv.Stoerung.Res_17 := FALSE;
   Schlamm_ED_Niv.Stoerung.Res_18 := FALSE;
   Schlamm_ED_Niv.Stoerung.Res_19 := FALSE;
   Schlamm_ED_Niv.Stoerung.Res_20 := FALSE;
   Schlamm_ED_Niv.Stoerung.Res_21 := FALSE;
   Schlamm_ED_Niv.Stoerung.Res_22 := FALSE;
   Schlamm_ED_Niv.Stoerung.Res_23 := FALSE;
   Schlamm_ED_Niv.Stoerung.Res_24 := FALSE;
   Schlamm_ED_Niv.Stoerung.Res_25 := FALSE;
   Schlamm_ED_Niv.Stoerung.Res_26 := FALSE;
   Schlamm_ED_Niv.Stoerung.Res_27 := FALSE;
   Schlamm_ED_Niv.Stoerung.Res_28 := FALSE;
   Schlamm_ED_Niv.Stoerung.Res_29 := FALSE;
   Schlamm_ED_Niv.Stoerung.Res_30 := FALSE;
   Schlamm_ED_Niv.Stoerung.Res_31 := FALSE;
   Schlamm_ED_Niv.MW_akt := 0.0;
   Schlamm_Besch_Niv.Status.BA_Nrm := TRUE;
   Schlamm_Besch_Niv.Status.BA_Frz := FALSE;
   Schlamm_Besch_Niv.Status.BA_EW := FALSE;
   Schlamm_Besch_Niv.Status.BA_Sim := FALSE;
   Schlamm_Besch_Niv.Status.BA_Wart := FALSE;
   Schlamm_Besch_Niv.Status.Frg_HH := FALSE;
   Schlamm_Besch_Niv.Status.Frg_H := FALSE;
   Schlamm_Besch_Niv.Status.Frg_L := FALSE;
   Schlamm_Besch_Niv.Status.Frg_LL := FALSE;
   Schlamm_Besch_Niv.Status.SB_MW_frz := FALSE;
   Schlamm_Besch_Niv.Status.SB_MW_EW := FALSE;
   Schlamm_Besch_Niv.Status.BM_MW_ok := TRUE;
   Schlamm_Besch_Niv.Status.BM_MW_frz := FALSE;
   Schlamm_Besch_Niv.Status.BM_MW_EW := FALSE;
   Schlamm_Besch_Niv.Status.BM_MW_Sim := FALSE;
   Schlamm_Besch_Niv.Status.BM_MW_nok := FALSE;
   Schlamm_Besch_Niv.Status.BM_MW_zw := FALSE;
   Schlamm_Besch_Niv.Status.GW_Sp_H := FALSE;
   Schlamm_Besch_Niv.Status.GW_Sp_L := FALSE;
   Schlamm_Besch_Niv.Status.Res_19 := FALSE;
   Schlamm_Besch_Niv.Status.Res_26 := FALSE;
   Schlamm_Besch_Niv.Status.Res_27 := FALSE;
   Schlamm_Besch_Niv.Status.Res_28 := FALSE;
   Schlamm_Besch_Niv.Status.Res_29 := FALSE;
   Schlamm_Besch_Niv.Status.Res_30 := FALSE;
   Schlamm_Besch_Niv.Status.Res_31 := FALSE;
   Schlamm_Besch_Niv.Status.Res_32 := FALSE;
   Schlamm_Besch_Niv.Status.Res_33 := FALSE;
   Schlamm_Besch_Niv.Status.Res_34 := FALSE;
   Schlamm_Besch_Niv.Status.BB_AutoOk := TRUE;
   Schlamm_Besch_Niv.Status.BB_SS := FALSE;
   Schlamm_Besch_Niv.Status.BB_SSnq := FALSE;
   Schlamm_Besch_Niv.Stoerung.St_allg := FALSE;
   Schlamm_Besch_Niv.Stoerung.St_4mA := FALSE;
   Schlamm_Besch_Niv.Stoerung.St_OF := FALSE;
   Schlamm_Besch_Niv.Stoerung.St_UF := FALSE;
   Schlamm_Besch_Niv.Stoerung.St_Kom_DP := FALSE;
   Schlamm_Besch_Niv.Stoerung.St_Kom_int := FALSE;
   Schlamm_Besch_Niv.Stoerung.St_int := FALSE;
   Schlamm_Besch_Niv.Stoerung.Res_7 := FALSE;
   Schlamm_Besch_Niv.Stoerung.GW_HH := FALSE;
   Schlamm_Besch_Niv.Stoerung.GW_H := FALSE;
   Schlamm_Besch_Niv.Stoerung.GW_L := FALSE;
   Schlamm_Besch_Niv.Stoerung.GW_LL := FALSE;
   Schlamm_Besch_Niv.Stoerung.Res_12 := FALSE;
   Schlamm_Besch_Niv.Stoerung.Res_13 := FALSE;
   Schlamm_Besch_Niv.Stoerung.Res_14 := FALSE;
   Schlamm_Besch_Niv.Stoerung.Res_15 := FALSE;
   Schlamm_Besch_Niv.Stoerung.Res_16 := FALSE;
   Schlamm_Besch_Niv.Stoerung.Res_17 := FALSE;
   Schlamm_Besch_Niv.Stoerung.Res_18 := FALSE;
   Schlamm_Besch_Niv.Stoerung.Res_19 := FALSE;
   Schlamm_Besch_Niv.Stoerung.Res_20 := FALSE;
   Schlamm_Besch_Niv.Stoerung.Res_21 := FALSE;
   Schlamm_Besch_Niv.Stoerung.Res_22 := FALSE;
   Schlamm_Besch_Niv.Stoerung.Res_23 := FALSE;
   Schlamm_Besch_Niv.Stoerung.Res_24 := FALSE;
   Schlamm_Besch_Niv.Stoerung.Res_25 := FALSE;
   Schlamm_Besch_Niv.Stoerung.Res_26 := FALSE;
   Schlamm_Besch_Niv.Stoerung.Res_27 := FALSE;
   Schlamm_Besch_Niv.Stoerung.Res_28 := FALSE;
   Schlamm_Besch_Niv.Stoerung.Res_29 := FALSE;
   Schlamm_Besch_Niv.Stoerung.Res_30 := FALSE;
   Schlamm_Besch_Niv.Stoerung.Res_31 := FALSE;
   Schlamm_Besch_Niv.MW_akt := 0.0;
   Schlamm_Besch_DF.Status.BA_Nrm := TRUE;
   Schlamm_Besch_DF.Status.BA_Frz := FALSE;
   Schlamm_Besch_DF.Status.BA_EW := FALSE;
   Schlamm_Besch_DF.Status.BA_Sim := FALSE;
   Schlamm_Besch_DF.Status.BA_Wart := FALSE;
   Schlamm_Besch_DF.Status.Frg_HH := FALSE;
   Schlamm_Besch_DF.Status.Frg_H := FALSE;
   Schlamm_Besch_DF.Status.Frg_L := FALSE;
   Schlamm_Besch_DF.Status.Frg_LL := FALSE;
   Schlamm_Besch_DF.Status.SB_MW_frz := FALSE;
   Schlamm_Besch_DF.Status.SB_MW_EW := FALSE;
   Schlamm_Besch_DF.Status.BM_MW_ok := TRUE;
   Schlamm_Besch_DF.Status.BM_MW_frz := FALSE;
   Schlamm_Besch_DF.Status.BM_MW_EW := FALSE;
   Schlamm_Besch_DF.Status.BM_MW_Sim := FALSE;
   Schlamm_Besch_DF.Status.BM_MW_nok := FALSE;
   Schlamm_Besch_DF.Status.BM_MW_zw := FALSE;
   Schlamm_Besch_DF.Status.GW_Sp_H := FALSE;
   Schlamm_Besch_DF.Status.GW_Sp_L := FALSE;
   Schlamm_Besch_DF.Status.Res_19 := FALSE;
   Schlamm_Besch_DF.Status.Res_26 := FALSE;
   Schlamm_Besch_DF.Status.Res_27 := FALSE;
   Schlamm_Besch_DF.Status.Res_28 := FALSE;
   Schlamm_Besch_DF.Status.Res_29 := FALSE;
   Schlamm_Besch_DF.Status.Res_30 := FALSE;
   Schlamm_Besch_DF.Status.Res_31 := FALSE;
   Schlamm_Besch_DF.Status.Res_32 := FALSE;
   Schlamm_Besch_DF.Status.Res_33 := FALSE;
   Schlamm_Besch_DF.Status.Res_34 := FALSE;
   Schlamm_Besch_DF.Status.BB_AutoOk := TRUE;
   Schlamm_Besch_DF.Status.BB_SS := FALSE;
   Schlamm_Besch_DF.Status.BB_SSnq := FALSE;
   Schlamm_Besch_DF.Stoerung.St_allg := FALSE;
   Schlamm_Besch_DF.Stoerung.St_4mA := FALSE;
   Schlamm_Besch_DF.Stoerung.St_OF := FALSE;
   Schlamm_Besch_DF.Stoerung.St_UF := FALSE;
   Schlamm_Besch_DF.Stoerung.St_Kom_DP := FALSE;
   Schlamm_Besch_DF.Stoerung.St_Kom_int := FALSE;
   Schlamm_Besch_DF.Stoerung.St_int := FALSE;
   Schlamm_Besch_DF.Stoerung.Res_7 := FALSE;
   Schlamm_Besch_DF.Stoerung.GW_HH := FALSE;
   Schlamm_Besch_DF.Stoerung.GW_H := FALSE;
   Schlamm_Besch_DF.Stoerung.GW_L := FALSE;
   Schlamm_Besch_DF.Stoerung.GW_LL := FALSE;
   Schlamm_Besch_DF.Stoerung.Res_12 := FALSE;
   Schlamm_Besch_DF.Stoerung.Res_13 := FALSE;
   Schlamm_Besch_DF.Stoerung.Res_14 := FALSE;
   Schlamm_Besch_DF.Stoerung.Res_15 := FALSE;
   Schlamm_Besch_DF.Stoerung.Res_16 := FALSE;
   Schlamm_Besch_DF.Stoerung.Res_17 := FALSE;
   Schlamm_Besch_DF.Stoerung.Res_18 := FALSE;
   Schlamm_Besch_DF.Stoerung.Res_19 := FALSE;
   Schlamm_Besch_DF.Stoerung.Res_20 := FALSE;
   Schlamm_Besch_DF.Stoerung.Res_21 := FALSE;
   Schlamm_Besch_DF.Stoerung.Res_22 := FALSE;
   Schlamm_Besch_DF.Stoerung.Res_23 := FALSE;
   Schlamm_Besch_DF.Stoerung.Res_24 := FALSE;
   Schlamm_Besch_DF.Stoerung.Res_25 := FALSE;
   Schlamm_Besch_DF.Stoerung.Res_26 := FALSE;
   Schlamm_Besch_DF.Stoerung.Res_27 := FALSE;
   Schlamm_Besch_DF.Stoerung.Res_28 := FALSE;
   Schlamm_Besch_DF.Stoerung.Res_29 := FALSE;
   Schlamm_Besch_DF.Stoerung.Res_30 := FALSE;
   Schlamm_Besch_DF.Stoerung.Res_31 := FALSE;
   Schlamm_Besch_DF.MW_akt := 0.00253176;
   Truebwasser_Niv.Status.BA_Nrm := TRUE;
   Truebwasser_Niv.Status.BA_Frz := FALSE;
   Truebwasser_Niv.Status.BA_EW := FALSE;
   Truebwasser_Niv.Status.BA_Sim := FALSE;
   Truebwasser_Niv.Status.BA_Wart := FALSE;
   Truebwasser_Niv.Status.Frg_HH := FALSE;
   Truebwasser_Niv.Status.Frg_H := FALSE;
   Truebwasser_Niv.Status.Frg_L := FALSE;
   Truebwasser_Niv.Status.Frg_LL := FALSE;
   Truebwasser_Niv.Status.SB_MW_frz := FALSE;
   Truebwasser_Niv.Status.SB_MW_EW := FALSE;
   Truebwasser_Niv.Status.BM_MW_ok := TRUE;
   Truebwasser_Niv.Status.BM_MW_frz := FALSE;
   Truebwasser_Niv.Status.BM_MW_EW := FALSE;
   Truebwasser_Niv.Status.BM_MW_Sim := FALSE;
   Truebwasser_Niv.Status.BM_MW_nok := FALSE;
   Truebwasser_Niv.Status.BM_MW_zw := FALSE;
   Truebwasser_Niv.Status.GW_Sp_H := FALSE;
   Truebwasser_Niv.Status.GW_Sp_L := FALSE;
   Truebwasser_Niv.Status.Res_19 := FALSE;
   Truebwasser_Niv.Status.Res_26 := FALSE;
   Truebwasser_Niv.Status.Res_27 := FALSE;
   Truebwasser_Niv.Status.Res_28 := FALSE;
   Truebwasser_Niv.Status.Res_29 := FALSE;
   Truebwasser_Niv.Status.Res_30 := FALSE;
   Truebwasser_Niv.Status.Res_31 := FALSE;
   Truebwasser_Niv.Status.Res_32 := FALSE;
   Truebwasser_Niv.Status.Res_33 := FALSE;
   Truebwasser_Niv.Status.Res_34 := FALSE;
   Truebwasser_Niv.Status.BB_AutoOk := TRUE;
   Truebwasser_Niv.Status.BB_SS := FALSE;
   Truebwasser_Niv.Status.BB_SSnq := FALSE;
   Truebwasser_Niv.Stoerung.St_allg := FALSE;
   Truebwasser_Niv.Stoerung.St_4mA := FALSE;
   Truebwasser_Niv.Stoerung.St_OF := FALSE;
   Truebwasser_Niv.Stoerung.St_UF := FALSE;
   Truebwasser_Niv.Stoerung.St_Kom_DP := FALSE;
   Truebwasser_Niv.Stoerung.St_Kom_int := FALSE;
   Truebwasser_Niv.Stoerung.St_int := FALSE;
   Truebwasser_Niv.Stoerung.Res_7 := FALSE;
   Truebwasser_Niv.Stoerung.GW_HH := FALSE;
   Truebwasser_Niv.Stoerung.GW_H := FALSE;
   Truebwasser_Niv.Stoerung.GW_L := FALSE;
   Truebwasser_Niv.Stoerung.GW_LL := FALSE;
   Truebwasser_Niv.Stoerung.Res_12 := FALSE;
   Truebwasser_Niv.Stoerung.Res_13 := FALSE;
   Truebwasser_Niv.Stoerung.Res_14 := FALSE;
   Truebwasser_Niv.Stoerung.Res_15 := FALSE;
   Truebwasser_Niv.Stoerung.Res_16 := FALSE;
   Truebwasser_Niv.Stoerung.Res_17 := FALSE;
   Truebwasser_Niv.Stoerung.Res_18 := FALSE;
   Truebwasser_Niv.Stoerung.Res_19 := FALSE;
   Truebwasser_Niv.Stoerung.Res_20 := FALSE;
   Truebwasser_Niv.Stoerung.Res_21 := FALSE;
   Truebwasser_Niv.Stoerung.Res_22 := FALSE;
   Truebwasser_Niv.Stoerung.Res_23 := FALSE;
   Truebwasser_Niv.Stoerung.Res_24 := FALSE;
   Truebwasser_Niv.Stoerung.Res_25 := FALSE;
   Truebwasser_Niv.Stoerung.Res_26 := FALSE;
   Truebwasser_Niv.Stoerung.Res_27 := FALSE;
   Truebwasser_Niv.Stoerung.Res_28 := FALSE;
   Truebwasser_Niv.Stoerung.Res_29 := FALSE;
   Truebwasser_Niv.Stoerung.Res_30 := FALSE;
   Truebwasser_Niv.Stoerung.Res_31 := FALSE;
   Truebwasser_Niv.MW_akt := 22.3247;
   Truebwasser_DF.Status.BA_Nrm := TRUE;
   Truebwasser_DF.Status.BA_Frz := FALSE;
   Truebwasser_DF.Status.BA_EW := FALSE;
   Truebwasser_DF.Status.BA_Sim := FALSE;
   Truebwasser_DF.Status.BA_Wart := FALSE;
   Truebwasser_DF.Status.Frg_HH := FALSE;
   Truebwasser_DF.Status.Frg_H := FALSE;
   Truebwasser_DF.Status.Frg_L := FALSE;
   Truebwasser_DF.Status.Frg_LL := FALSE;
   Truebwasser_DF.Status.SB_MW_frz := FALSE;
   Truebwasser_DF.Status.SB_MW_EW := FALSE;
   Truebwasser_DF.Status.BM_MW_ok := TRUE;
   Truebwasser_DF.Status.BM_MW_frz := FALSE;
   Truebwasser_DF.Status.BM_MW_EW := FALSE;
   Truebwasser_DF.Status.BM_MW_Sim := FALSE;
   Truebwasser_DF.Status.BM_MW_nok := FALSE;
   Truebwasser_DF.Status.BM_MW_zw := FALSE;
   Truebwasser_DF.Status.GW_Sp_H := FALSE;
   Truebwasser_DF.Status.GW_Sp_L := FALSE;
   Truebwasser_DF.Status.Res_19 := FALSE;
   Truebwasser_DF.Status.Res_26 := FALSE;
   Truebwasser_DF.Status.Res_27 := FALSE;
   Truebwasser_DF.Status.Res_28 := FALSE;
   Truebwasser_DF.Status.Res_29 := FALSE;
   Truebwasser_DF.Status.Res_30 := FALSE;
   Truebwasser_DF.Status.Res_31 := FALSE;
   Truebwasser_DF.Status.Res_32 := FALSE;
   Truebwasser_DF.Status.Res_33 := FALSE;
   Truebwasser_DF.Status.Res_34 := FALSE;
   Truebwasser_DF.Status.BB_AutoOk := TRUE;
   Truebwasser_DF.Status.BB_SS := FALSE;
   Truebwasser_DF.Status.BB_SSnq := FALSE;
   Truebwasser_DF.Stoerung.St_allg := FALSE;
   Truebwasser_DF.Stoerung.St_4mA := FALSE;
   Truebwasser_DF.Stoerung.St_OF := FALSE;
   Truebwasser_DF.Stoerung.St_UF := FALSE;
   Truebwasser_DF.Stoerung.St_Kom_DP := FALSE;
   Truebwasser_DF.Stoerung.St_Kom_int := FALSE;
   Truebwasser_DF.Stoerung.St_int := FALSE;
   Truebwasser_DF.Stoerung.Res_7 := FALSE;
   Truebwasser_DF.Stoerung.GW_HH := FALSE;
   Truebwasser_DF.Stoerung.GW_H := FALSE;
   Truebwasser_DF.Stoerung.GW_L := FALSE;
   Truebwasser_DF.Stoerung.GW_LL := FALSE;
   Truebwasser_DF.Stoerung.Res_12 := FALSE;
   Truebwasser_DF.Stoerung.Res_13 := FALSE;
   Truebwasser_DF.Stoerung.Res_14 := FALSE;
   Truebwasser_DF.Stoerung.Res_15 := FALSE;
   Truebwasser_DF.Stoerung.Res_16 := FALSE;
   Truebwasser_DF.Stoerung.Res_17 := FALSE;
   Truebwasser_DF.Stoerung.Res_18 := FALSE;
   Truebwasser_DF.Stoerung.Res_19 := FALSE;
   Truebwasser_DF.Stoerung.Res_20 := FALSE;
   Truebwasser_DF.Stoerung.Res_21 := FALSE;
   Truebwasser_DF.Stoerung.Res_22 := FALSE;
   Truebwasser_DF.Stoerung.Res_23 := FALSE;
   Truebwasser_DF.Stoerung.Res_24 := FALSE;
   Truebwasser_DF.Stoerung.Res_25 := FALSE;
   Truebwasser_DF.Stoerung.Res_26 := FALSE;
   Truebwasser_DF.Stoerung.Res_27 := FALSE;
   Truebwasser_DF.Stoerung.Res_28 := FALSE;
   Truebwasser_DF.Stoerung.Res_29 := FALSE;
   Truebwasser_DF.Stoerung.Res_30 := FALSE;
   Truebwasser_DF.Stoerung.Res_31 := FALSE;
   Truebwasser_DF.MW_akt := -0.001695375;
   Zulauf_SF_Niv.Status.BA_Nrm := TRUE;
   Zulauf_SF_Niv.Status.BA_Frz := FALSE;
   Zulauf_SF_Niv.Status.BA_EW := FALSE;
   Zulauf_SF_Niv.Status.BA_Sim := FALSE;
   Zulauf_SF_Niv.Status.BA_Wart := FALSE;
   Zulauf_SF_Niv.Status.Frg_HH := FALSE;
   Zulauf_SF_Niv.Status.Frg_H := FALSE;
   Zulauf_SF_Niv.Status.Frg_L := FALSE;
   Zulauf_SF_Niv.Status.Frg_LL := FALSE;
   Zulauf_SF_Niv.Status.SB_MW_frz := FALSE;
   Zulauf_SF_Niv.Status.SB_MW_EW := FALSE;
   Zulauf_SF_Niv.Status.BM_MW_ok := TRUE;
   Zulauf_SF_Niv.Status.BM_MW_frz := FALSE;
   Zulauf_SF_Niv.Status.BM_MW_EW := FALSE;
   Zulauf_SF_Niv.Status.BM_MW_Sim := FALSE;
   Zulauf_SF_Niv.Status.BM_MW_nok := FALSE;
   Zulauf_SF_Niv.Status.BM_MW_zw := FALSE;
   Zulauf_SF_Niv.Status.GW_Sp_H := FALSE;
   Zulauf_SF_Niv.Status.GW_Sp_L := FALSE;
   Zulauf_SF_Niv.Status.Res_19 := FALSE;
   Zulauf_SF_Niv.Status.Res_26 := FALSE;
   Zulauf_SF_Niv.Status.Res_27 := FALSE;
   Zulauf_SF_Niv.Status.Res_28 := FALSE;
   Zulauf_SF_Niv.Status.Res_29 := FALSE;
   Zulauf_SF_Niv.Status.Res_30 := FALSE;
   Zulauf_SF_Niv.Status.Res_31 := FALSE;
   Zulauf_SF_Niv.Status.Res_32 := FALSE;
   Zulauf_SF_Niv.Status.Res_33 := FALSE;
   Zulauf_SF_Niv.Status.Res_34 := FALSE;
   Zulauf_SF_Niv.Status.BB_AutoOk := TRUE;
   Zulauf_SF_Niv.Status.BB_SS := FALSE;
   Zulauf_SF_Niv.Status.BB_SSnq := FALSE;
   Zulauf_SF_Niv.Stoerung.St_allg := FALSE;
   Zulauf_SF_Niv.Stoerung.St_4mA := FALSE;
   Zulauf_SF_Niv.Stoerung.St_OF := FALSE;
   Zulauf_SF_Niv.Stoerung.St_UF := FALSE;
   Zulauf_SF_Niv.Stoerung.St_Kom_DP := FALSE;
   Zulauf_SF_Niv.Stoerung.St_Kom_int := FALSE;
   Zulauf_SF_Niv.Stoerung.St_int := FALSE;
   Zulauf_SF_Niv.Stoerung.Res_7 := FALSE;
   Zulauf_SF_Niv.Stoerung.GW_HH := FALSE;
   Zulauf_SF_Niv.Stoerung.GW_H := FALSE;
   Zulauf_SF_Niv.Stoerung.GW_L := FALSE;
   Zulauf_SF_Niv.Stoerung.GW_LL := FALSE;
   Zulauf_SF_Niv.Stoerung.Res_12 := FALSE;
   Zulauf_SF_Niv.Stoerung.Res_13 := FALSE;
   Zulauf_SF_Niv.Stoerung.Res_14 := FALSE;
   Zulauf_SF_Niv.Stoerung.Res_15 := FALSE;
   Zulauf_SF_Niv.Stoerung.Res_16 := FALSE;
   Zulauf_SF_Niv.Stoerung.Res_17 := FALSE;
   Zulauf_SF_Niv.Stoerung.Res_18 := FALSE;
   Zulauf_SF_Niv.Stoerung.Res_19 := FALSE;
   Zulauf_SF_Niv.Stoerung.Res_20 := FALSE;
   Zulauf_SF_Niv.Stoerung.Res_21 := FALSE;
   Zulauf_SF_Niv.Stoerung.Res_22 := FALSE;
   Zulauf_SF_Niv.Stoerung.Res_23 := FALSE;
   Zulauf_SF_Niv.Stoerung.Res_24 := FALSE;
   Zulauf_SF_Niv.Stoerung.Res_25 := FALSE;
   Zulauf_SF_Niv.Stoerung.Res_26 := FALSE;
   Zulauf_SF_Niv.Stoerung.Res_27 := FALSE;
   Zulauf_SF_Niv.Stoerung.Res_28 := FALSE;
   Zulauf_SF_Niv.Stoerung.Res_29 := FALSE;
   Zulauf_SF_Niv.Stoerung.Res_30 := FALSE;
   Zulauf_SF_Niv.Stoerung.Res_31 := FALSE;
   Zulauf_SF_Niv.MW_akt := 0.0;
   Ablauf_NOx.Status.BA_Nrm := TRUE;
   Ablauf_NOx.Status.BA_Frz := FALSE;
   Ablauf_NOx.Status.BA_EW := FALSE;
   Ablauf_NOx.Status.BA_Sim := FALSE;
   Ablauf_NOx.Status.BA_Wart := FALSE;
   Ablauf_NOx.Status.Frg_HH := FALSE;
   Ablauf_NOx.Status.Frg_H := FALSE;
   Ablauf_NOx.Status.Frg_L := FALSE;
   Ablauf_NOx.Status.Frg_LL := FALSE;
   Ablauf_NOx.Status.SB_MW_frz := FALSE;
   Ablauf_NOx.Status.SB_MW_EW := FALSE;
   Ablauf_NOx.Status.BM_MW_ok := TRUE;
   Ablauf_NOx.Status.BM_MW_frz := FALSE;
   Ablauf_NOx.Status.BM_MW_EW := FALSE;
   Ablauf_NOx.Status.BM_MW_Sim := FALSE;
   Ablauf_NOx.Status.BM_MW_nok := FALSE;
   Ablauf_NOx.Status.BM_MW_zw := FALSE;
   Ablauf_NOx.Status.GW_Sp_H := FALSE;
   Ablauf_NOx.Status.GW_Sp_L := FALSE;
   Ablauf_NOx.Status.Res_19 := FALSE;
   Ablauf_NOx.Status.Res_26 := FALSE;
   Ablauf_NOx.Status.Res_27 := FALSE;
   Ablauf_NOx.Status.Res_28 := FALSE;
   Ablauf_NOx.Status.Res_29 := FALSE;
   Ablauf_NOx.Status.Res_30 := FALSE;
   Ablauf_NOx.Status.Res_31 := FALSE;
   Ablauf_NOx.Status.Res_32 := FALSE;
   Ablauf_NOx.Status.Res_33 := FALSE;
   Ablauf_NOx.Status.Res_34 := FALSE;
   Ablauf_NOx.Status.BB_AutoOk := TRUE;
   Ablauf_NOx.Status.BB_SS := FALSE;
   Ablauf_NOx.Status.BB_SSnq := FALSE;
   Ablauf_NOx.Stoerung.St_allg := FALSE;
   Ablauf_NOx.Stoerung.St_4mA := FALSE;
   Ablauf_NOx.Stoerung.St_OF := FALSE;
   Ablauf_NOx.Stoerung.St_UF := FALSE;
   Ablauf_NOx.Stoerung.St_Kom_DP := FALSE;
   Ablauf_NOx.Stoerung.St_Kom_int := FALSE;
   Ablauf_NOx.Stoerung.St_int := FALSE;
   Ablauf_NOx.Stoerung.Res_7 := FALSE;
   Ablauf_NOx.Stoerung.GW_HH := FALSE;
   Ablauf_NOx.Stoerung.GW_H := FALSE;
   Ablauf_NOx.Stoerung.GW_L := FALSE;
   Ablauf_NOx.Stoerung.GW_LL := FALSE;
   Ablauf_NOx.Stoerung.Res_12 := FALSE;
   Ablauf_NOx.Stoerung.Res_13 := FALSE;
   Ablauf_NOx.Stoerung.Res_14 := FALSE;
   Ablauf_NOx.Stoerung.Res_15 := FALSE;
   Ablauf_NOx.Stoerung.Res_16 := FALSE;
   Ablauf_NOx.Stoerung.Res_17 := FALSE;
   Ablauf_NOx.Stoerung.Res_18 := FALSE;
   Ablauf_NOx.Stoerung.Res_19 := FALSE;
   Ablauf_NOx.Stoerung.Res_20 := FALSE;
   Ablauf_NOx.Stoerung.Res_21 := FALSE;
   Ablauf_NOx.Stoerung.Res_22 := FALSE;
   Ablauf_NOx.Stoerung.Res_23 := FALSE;
   Ablauf_NOx.Stoerung.Res_24 := FALSE;
   Ablauf_NOx.Stoerung.Res_25 := FALSE;
   Ablauf_NOx.Stoerung.Res_26 := FALSE;
   Ablauf_NOx.Stoerung.Res_27 := FALSE;
   Ablauf_NOx.Stoerung.Res_28 := FALSE;
   Ablauf_NOx.Stoerung.Res_29 := FALSE;
   Ablauf_NOx.Stoerung.Res_30 := FALSE;
   Ablauf_NOx.Stoerung.Res_31 := FALSE;
   Ablauf_NOx.MW_akt := 1.462996;
   Ablauf_PO4.Status.BA_Nrm := TRUE;
   Ablauf_PO4.Status.BA_Frz := FALSE;
   Ablauf_PO4.Status.BA_EW := FALSE;
   Ablauf_PO4.Status.BA_Sim := FALSE;
   Ablauf_PO4.Status.BA_Wart := FALSE;
   Ablauf_PO4.Status.Frg_HH := FALSE;
   Ablauf_PO4.Status.Frg_H := FALSE;
   Ablauf_PO4.Status.Frg_L := FALSE;
   Ablauf_PO4.Status.Frg_LL := FALSE;
   Ablauf_PO4.Status.SB_MW_frz := FALSE;
   Ablauf_PO4.Status.SB_MW_EW := FALSE;
   Ablauf_PO4.Status.BM_MW_ok := TRUE;
   Ablauf_PO4.Status.BM_MW_frz := FALSE;
   Ablauf_PO4.Status.BM_MW_EW := FALSE;
   Ablauf_PO4.Status.BM_MW_Sim := FALSE;
   Ablauf_PO4.Status.BM_MW_nok := FALSE;
   Ablauf_PO4.Status.BM_MW_zw := FALSE;
   Ablauf_PO4.Status.GW_Sp_H := FALSE;
   Ablauf_PO4.Status.GW_Sp_L := FALSE;
   Ablauf_PO4.Status.Res_19 := FALSE;
   Ablauf_PO4.Status.Res_26 := FALSE;
   Ablauf_PO4.Status.Res_27 := FALSE;
   Ablauf_PO4.Status.Res_28 := FALSE;
   Ablauf_PO4.Status.Res_29 := FALSE;
   Ablauf_PO4.Status.Res_30 := FALSE;
   Ablauf_PO4.Status.Res_31 := FALSE;
   Ablauf_PO4.Status.Res_32 := FALSE;
   Ablauf_PO4.Status.Res_33 := FALSE;
   Ablauf_PO4.Status.Res_34 := FALSE;
   Ablauf_PO4.Status.BB_AutoOk := TRUE;
   Ablauf_PO4.Status.BB_SS := FALSE;
   Ablauf_PO4.Status.BB_SSnq := FALSE;
   Ablauf_PO4.Stoerung.St_allg := FALSE;
   Ablauf_PO4.Stoerung.St_4mA := FALSE;
   Ablauf_PO4.Stoerung.St_OF := FALSE;
   Ablauf_PO4.Stoerung.St_UF := FALSE;
   Ablauf_PO4.Stoerung.St_Kom_DP := FALSE;
   Ablauf_PO4.Stoerung.St_Kom_int := FALSE;
   Ablauf_PO4.Stoerung.St_int := FALSE;
   Ablauf_PO4.Stoerung.Res_7 := FALSE;
   Ablauf_PO4.Stoerung.GW_HH := FALSE;
   Ablauf_PO4.Stoerung.GW_H := FALSE;
   Ablauf_PO4.Stoerung.GW_L := FALSE;
   Ablauf_PO4.Stoerung.GW_LL := FALSE;
   Ablauf_PO4.Stoerung.Res_12 := FALSE;
   Ablauf_PO4.Stoerung.Res_13 := FALSE;
   Ablauf_PO4.Stoerung.Res_14 := FALSE;
   Ablauf_PO4.Stoerung.Res_15 := FALSE;
   Ablauf_PO4.Stoerung.Res_16 := FALSE;
   Ablauf_PO4.Stoerung.Res_17 := FALSE;
   Ablauf_PO4.Stoerung.Res_18 := FALSE;
   Ablauf_PO4.Stoerung.Res_19 := FALSE;
   Ablauf_PO4.Stoerung.Res_20 := FALSE;
   Ablauf_PO4.Stoerung.Res_21 := FALSE;
   Ablauf_PO4.Stoerung.Res_22 := FALSE;
   Ablauf_PO4.Stoerung.Res_23 := FALSE;
   Ablauf_PO4.Stoerung.Res_24 := FALSE;
   Ablauf_PO4.Stoerung.Res_25 := FALSE;
   Ablauf_PO4.Stoerung.Res_26 := FALSE;
   Ablauf_PO4.Stoerung.Res_27 := FALSE;
   Ablauf_PO4.Stoerung.Res_28 := FALSE;
   Ablauf_PO4.Stoerung.Res_29 := FALSE;
   Ablauf_PO4.Stoerung.Res_30 := FALSE;
   Ablauf_PO4.Stoerung.Res_31 := FALSE;
   Ablauf_PO4.MW_akt := 2.768842;

END_DATA_BLOCK

DATA_BLOCK "DB115_MW_Bef_PLS"
{ S7_Optimized_Access := 'FALSE' }
VERSION : 0.1
NON_RETAIN
   STRUCT
      Zulauf_AR_Niv : "T_MW_BEF";   // Zulauf - Pumpwerk "Alter Rechen" - Niveau
      Zulauf_AR_Temp : "T_MW_BEF";   // Zulauf - Pumpwerk "Alter Rechen" - Temperatur
      Zulauf_AR_DF : "T_MW_BEF";   // Zulauf - Pumpwerk "Alter Rechen" - Durchfluss
      BB1_AS1_SS : "T_MW_BEF";   // Becken 1 - Ablaufschieber 1 - Schieberstellung
      BB1_AS2_SS : "T_MW_BEF";   // Becken 1 - Ablaufschieber 2 - Schieberstellung
      BB2_AS1_SS : "T_MW_BEF";   // Becken 2 - Ablaufschieber 1 - Schieberstellung
      BB2_AS2_SS : "T_MW_BEF";   // Becken 2 - Ablaufschieber 2 - Schieberstellung
      BB1_O2 : "T_MW_BEF";   // Becken 1 - O2-Gehalt
      BB1_Temp : "T_MW_BEF";   // Becken 1 - Temperatur
      BB2_O2 : "T_MW_BEF";   // Becken 2 - O2-Gehalt
      BB2_Temp : "T_MW_BEF";   // Becken 2 - Temperatur
      BB1_DF : "T_MW_BEF";   // Becken 1 - Ablauf - Durchfluss
      BB2_DF : "T_MW_BEF";   // Becken 2 - Ablauf - Durchfluss
      Zulauf_Niv : "T_MW_BEF";   // Zulauf - Vorlagebehälter - Niveau
      Zulauf_DF : "T_MW_BEF";   // Zulauf - Rechen - Durchfluss
      Verteiler_pH : "T_MW_BEF";   // Zulauf - Verteiler - pH-Wert
      Verteiler_O2 : "T_MW_BEF";   // Zulauf - Verteiler  - O2-Gehalt
      Verteiler_Temp : "T_MW_BEF";   // Zulauf - Verteiler - Temperatur
      BB_UeSS_DF : "T_MW_BEF";   // Becken 1+2 - Ablauf ÜSS - Durchfluss
      Ablauf_DF : "T_MW_BEF";   // Ablauf - Durchfluss
      Ablauf_pH : "T_MW_BEF";   // Ablauf - pH-Wert
      Ablauf_O2 : "T_MW_BEF";   // Ablauf - O2-Gehalt
      Ablauf_Temp : "T_MW_BEF";   // Ablauf - Temperatur
      Schlamm_ED_Niv : "T_MW_BEF";   // Schlamm - Eindicker - Niveau
      Schlamm_Besch_Niv : "T_MW_BEF";   // Schlamm - Beschickung - Niveau
      Schlamm_Besch_DF : "T_MW_BEF";   // Schlamm - Beschickung - Durchfluss
      Truebwasser_Niv : "T_MW_BEF";   // Trübwasserpumpwerk - Niveau
      Truebwasser_DF : "T_MW_BEF";   // Trübwasserpumpwerk - Durchfluss
      Zulauf_SF_Niv : "T_MW_BEF";   // Zulauf - Sandfang - Niveau
      Ablauf_NOx : "T_MW_BEF";   // Ablauf - Dortmundbrunnen - Nitratmessung
      Ablauf_PO4 : "T_MW_BEF";   // Ablauf - Dortmundbrunnen - Phosphatmessung
      Umwelt_WG : "T_MW_BEF";   // Wetterstation - Windgeschwindigkeit
      Umwelt_WR : "T_MW_BEF";   // Wetterstation - Windrichtung
      Umwelt_LDr : "T_MW_BEF";   // Wetterstation - Luftdruck
      Umwelt_LF : "T_MW_BEF";   // Wetterstation - Luftfeuchtigkeit
      Umwelt_T : "T_MW_BEF";   // Wetterstation - Temperatur
      Ablauf_LF : "T_MW_BEF";   // Ablauf - Leitfähigkeit
   END_STRUCT;


